(* CODESYS project 3_1_5_4.library
   Company: StroemHansen
   Title: SH_Light
   Description: Adds override function to
      FB_TwoVal_SelectOne_RTrigChange
      
      Fixes bugs in
      FB_FoldingDoorCtrl_2Pcs
      
      Replaces 3.1.5.3
   Placeholder: SH_Light
   Author: Jonas Justsen
   Version: 3.1.5.4

Project tree, tasks and I/O mapping:
  libraries: Tc2_ModbusSrv, * (Beckhoff Automation GmbH); Tc2_Standard, * (Beckhoff Automation GmbH); Tc2_System, * (Beckhoff Automation GmbH); Tc2_Utilities, * (Beckhoff Automation GmbH); Tc3_DALI, * (Beckhoff Automation GmbH)
  DUTs/
    data type E_OnMode
    data type ST_DALI_Energy
    data type ST_DALI_GrpAssignment
    data type ST_DALI_NIKOP46SetupData
    data type ST_DALI_RoomSetup
    data type ST_DALI_Sensor
    data type ST_DALI_SensorScaleMode
    data type ST_DALIButton
    data type ST_GlamoxSetup
    data type ST_GroupSort
    data type ST_LgtCmd
    data type ST_LiveData
    data type ST_LunatoneMCSetup
    data type ST_NeighborIP
    data type ST_RoomDataPLC
    data type ST_TuneData_EX
  GVLs/
    global variables DALI_Param
    global variables GVL_DALI
    global variables GVL_DALI_LatestError
  POUs/
    DALI/
      Ballast/
        function F_fDALICurve [ST]
        function F_fDALICurveRev [ST]
        function block FB_DALI_Diag [ST]: A_DALICmdAddressing, A_DALICmdAddToGroup, A_DALICmdQueryGroups, A_DALICmdQueryLampFailure, A_DALICmdQueryMissingShortAddress, A_DALICmdQueryStatus, A_ResetRoutine, A_SetAddressesToGroups, ipDALICommunication, TrySetCommunication
        function block FB_DALI_EnergyDataManagement [ST]
        function block FB_DALI_EnergyReporting [ST]: A_DALI252QueryActiveEnergy, A_DALI252QueryActiveEnergyLoadside, A_DALI252QueryActivePower, A_DALI252QueryActivePowerLoadside, A_DALI252QueryApparentEnergy, A_DALI252QueryApparentPower, A_DALI253QueryControlGearOperatingTime, A_DALI253QueryControlGearStartCounter, A_DALI253QueryLightSourceStartCounter, A_ResetRoutine, ipDALICommunication, TrySetCommunication
        function block FB_DALILgtActr_EX [ST]: A_DALICmdDirectArcPowerControl, A_DALICmdDirectArcPowerControl_Sttup, A_DALICmdDown, A_DALICmdOff, A_DALICmdQueryActualLevel, A_DALICmdQueryMaxLevel, A_DALICmdQueryMinLevel, A_DALICmdQueryPhysicalMinLevel, A_DALICmdRecallMaxLevel, A_DALICmdRecallMinLevel, A_DALICmdSetFadeRate, A_DALICmdSetFadeTime, A_DALICmdSetMaxLevel_CmdSt, A_DALICmdSetMaxLevel_Input, A_DALICmdSetMinLevel_CmdSt, A_DALICmdSetMinLevel_Input, A_DALICmdStepDown, A_DALICmdStepUp, A_DALICmdUp, A_ResetRoutine, ipDALICommunication, TrySetCommunication
        function block FB_DALILgtActr_Simple [ST]: A_DALICmdDirectArcPowerControl, A_DALICmdDirectArcPowerControl_Sttup, A_DALICmdDown, A_DALICmdOff, A_DALICmdQueryActualLevel, A_DALICmdQueryMaxLevel, A_DALICmdQueryMinLevel, A_DALICmdQueryPhysicalMinLevel, A_DALICmdRecallMaxLevel, A_DALICmdRecallMinLevel, A_DALICmdStepDown, A_DALICmdStepUp, A_DALICmdUp, A_ResetRoutine, ipDALICommunication, TrySetCommunication
        function block FB_DALILgtCfg [ST]: A_DALICmdQueryActualLevel, A_DALICmdQueryMaxLevel, A_DALICmdQueryMinLevel, A_DALICmdQueryPhysicalMinLevel, A_DALICmdSetFadeRate, A_DALICmdSetFadeTime, A_DALICmdSetMaxLevel_CmdSt, A_DALICmdSetMaxLevel_Input, A_DALICmdSetMinLevel_CmdSt, A_DALICmdSetMinLevel_Input, A_ResetRoutine, ipDALICommunication, TrySetCommunication
        function block FB_Light_Ballast [ST]: M_PrimBallast, M_SecBallast, M_SuplBallast
        function block FB_Light_SingleBallast [ST]: M_Ballast
        function block FB_MasterSelector [ST]
      Color (DT8)/
        function F_iColorMix [ST]
        function block FB_DALI_RGBWAFLight [ST]: A_DALICmdActivate_DT8, A_DALICmdTemporaryRGBDimlevel, A_DALICmdTemporaryRGBWAFControl, A_DALICmdTemporaryWAFDimlevel, A_DALIQueryColourValueAmber, A_DALIQueryColourValueBlue, A_DALIQueryColourValueFreeColor, A_DALIQueryColourValueGreen, A_DALIQueryColourValueRed, A_DALIQueryColourValueWhite, A_ResetRoutine, ipDALICommunication, TrySetCommunication
        function block FB_DALI_TcColorLight [ST]: A_DALICmdActivate_DT8, A_DALICmdSetColourTemperatureTc, A_DALIQueryColourStatus, A_DALIQueryColourTc, A_ResetRoutine, ipDALICommunication, TrySetCommunication
      DALI_Devices/
        BEG/
          function block FB_BEG_PD2N_1Pcs [ST]: A_BEG_PD2N_1
        ESYLux/
          Flat/
            function block FB_DALI_ESYLuxFlat_1Pcs [ST]: A_ESYLux_1
          function block FB_DALI_ESYLux_1Pcs [ST]: A_ESYLux_1
          function block FB_DALI_ESYLux_2Pcs [ST]: A_ESYLux_2Pcs
          function block FB_DALI_ESYLux_3Pcs [ST]: A_ESYLux_3Pcs
          function block FB_DALI_ESYLux_4Pcs [ST]: A_ESYLux_4Pcs
          function block FB_DALI_ESYLux_5Pcs [ST]: A_ESYLux_5Pcs
          function block FB_DALI_ESYLux_6Pcs [ST]: A_ESYLux_6Pcs
        Glamox/
          function block FB_DALI_GlamoxButtons [ST]: A_Sort_Event_Button1, A_Sort_Event_Button2, A_Sort_Event_Button3, A_Sort_Event_Button4, A_Sort_Event_Button5, A_Sort_Event_Button6, A_Sort_Event_Button7, A_Sort_Event_Button8
        Lunatone/
          function block FB_DALI_Lunatone_MC2_OLD [ST]: A_LunatonButton
          function block FB_DALI_Lunatone_ROT [ST]: A_LunatonRotation
          function block FB_DALI_LunatoneMC [ST]: A_Sort_Event_Button1, A_Sort_Event_Button2, A_Sort_Event_Button3, A_Sort_Event_Button4
        NIKO/
          function block FB_NIKO_P46xx_10Pcs [ST]: A_NIKO_P46xx
          function block FB_NIKO_P46xx_1Pcs [ST]: A_NIKO_P46xx_1
          function block FB_NIKO_P46xx_2Pcs [ST]: A_NIKO_P46xx
          function block FB_NIKO_P46xx_3Pcs [ST]: A_NIKO_P46xx
          function block FB_NIKO_P46xx_4Pcs [ST]: A_NIKO_P46xx
          function block FB_NIKO_P46xx_5Pcs [ST]: A_NIKO_P46xx
          function block FB_NIKO_P46xx_6Pcs [ST]: A_NIKO_P46xx
          function block FB_NIKO_P46xx_7Pcs [ST]: A_NIKO_P46xx
          function block FB_NIKO_P46xx_8Pcs [ST]: A_NIKO_P46xx
          function block FB_NIKO_P46xx_9Pcs [ST]: A_NIKO_P46xx
      FBs/
        function block FB_Short [ST]
        function block FB_ValTrig_F [ST]
      FUNs/
        function F_fScale [ST]
        function F_lrScale_EX [ST]
      Lunatone/
        function block FB_DALI_Lunatone_ROT_D2I_Mode [ST]: bEnablePosition, eEventPriorityPosition, nDeadtimerPosition, nReportTimePosition, bEnablePushButton, eEventPriorityButton, nDoubleTimerPushButton, nEventFilterPushButton, nRepeatTimerPushButton, nShortTimerPushButton, nStuckTimerPushButton, bEnableRotation, eEventPriorityRotation, nEventFilterRotation, CheckParameters, FB_init, ipDALICommunication, ParameterChanged, SetCommunication
        data type ST_ROT
      MUX/
        Timing/
          function block FB_MinOnMinOffTime [ST]
      Operators/
        function block FB_BA_Swi [ST]
        function block FB_BA_ValTrigF [ST]
        function block FB_Click [ST]
        function block FB_FileCopy [ST]
        function block FB_Ramper [ST]
      Power Control/
        function block FB_AutoTune_TcBA_EX [ST]
        function block FB_DirectLight_1Group [ST]
        function block FB_LightCtrl_1Group [ST]
        function block FB_LightCtrl_1Group_ [ST]
        function block FB_LightCtrl_1Group_OLD [ST]
        function block FB_LightCtrl_2Groups [ST]
        function block FB_LightCtrl_2Groups_Action [ST]: A_Auto, A_Manuel, A_Tuning
        function block FB_LightSwitch [ST]: A_BA_LgtSwi_ResetCommands, A_BA_LgtSwi_WaitToReset
        function block FB_SearchStartUpLevel_EX [ST]
    Folding_Doors/
      function block FB_ConnectRooms_3Pcs [ST]: A_ButtonLogic, A_OverrideLogic, A_SensorLogic
      function block FB_ConnectRooms_xPcs [ST]: A_ButtonLogic, A_OverrideLogic, A_SensorLogic
      function block FB_FoldingDoor [ST]: A_ButtonLogic, A_OverrideLogic, A_SensorLogic
      function block FB_FoldingDoorCtrl_2Pcs [ST]: A_State0, A_State1, A_State2, A_State3
    Internals/
      function block FB_FunctionType_A [ST]
    Misc/
      function F_CltsEveryBool [ST]
      function block FB_ClockPulse [ST]
      function block FB_CountOnHours [ST]
      function block FB_TwoVal_SelectOne_RTrigChange [ST]
    Modbus/
      function block FB_ReadAHPirData [ST]
    Scheduling/
      function block FB_TODScheduling [ST]
    Templates/
      function block FB_Light_Type_A [ST]: A_DaliUpdate, A_RoomFct, A_TuningProcess
      function block FB_Light_Type_B [ST]: A_DaliUpdate, A_RoomFct, A_TuningProcess
  Project Information/
    function F_GetCompany [ST]
    function F_GetTitle [ST]
    function F_GetVersion [ST]
  Version/
    global variables Global_Version
  VISUs/
*)

// DUTs/E_OnMode
TYPE E_OnMode :
(	e_ClMaxVal 				:= 0,
	e_ClMinVal 				:= 1,
	e_ClOnVal 				:= 2,
	e_ClRstVal 				:= 3
);END_TYPE

// DUTs/ST_DALI_Energy
TYPE ST_DALI_Energy :
STRUCT
	fActiveEnergy				: LREAL;
	fActiveEnergyLoadside		: LREAL;
	fActivePower				: LREAL;
	fActivePowerLoadside 		: LREAL;
	fApparentEnergy 			: LREAL;
	fApparentPower 				: LREAL;
	nControlGearOperatingTime  	: UDINT;
	nControlGearStartCounter   	: UDINT;	
	nLightSourceStartCounter   	: UDINT;
	bHasEnergyData				: BOOL;
END_STRUCT
END_TYPE

// DUTs/ST_DALI_GrpAssignment
TYPE ST_DALI_GrpAssignment :
STRUCT
	bLampPresentInNetwork: BOOL;
	bFaultOnDALIBallast : BOOL;
	bLampFailur : BOOL;
	bLampPowerOn : BOOL;
	bLimitErrVal : BOOL;
	bDimmingActive: BOOL;
	bResetState	: BOOL;
	bShortAddrMissing: BOOL;
	bPowerSupplyWasEnabled: BOOL;
	nGroups	: WORD; 	
END_STRUCT
END_TYPE

// DUTs/ST_DALI_NIKOP46SetupData
TYPE ST_DALI_NIKOP46SetupData :
STRUCT
	bInitialize						:	BOOL := TRUE;
	bQueryInputValueOccupancy			:	BOOL ;
	bQueryInputValueBrightness		:	BOOL ;
	//Parameters Motion
	bEnableInstanceOccupancy			:	BOOL := TRUE;
	eEventPriorityOccupancy			: 	E_DALIEventPriority := E_DALIEVENTPRIORITY.Middle;
	nReportTimerOccupancy				:	BYTE := 120; // Value in s, Preset manufacturer value
	nDeadtimeTimerOccupancy			:	WORD := 100; // Value in ms, Predefined Value of DALI Standard
	nHoldTimerOccupancy				:	WORD := 120; // Value in s. 
	bCancelHoldTimeOccupancy			:	BOOL := FALSE;
	nSensitivityPIRSegmentA			:	BYTE := 16#01; // Preset manufacturer value: 0 = Max, 1 = High, 2 = Low, 3 = Min, 4 = Off
	nSensitivityPIRSegmentB			:	BYTE := 16#01; // Preset manufacturer value: 0 = Max, 1 = High, 2 = Low, 3 = Min, 4 = Off
	nSensitivityPIRSegmentC			:	BYTE := 16#01; // Preset manufacturer value: 0 = Max, 1 = High, 2 = Low, 3 = Min, 4 = Off
	//Parameters Brightness
	bEnableInstanceBrightness		:	BOOL := TRUE;
	eEventPriorityBrightness		: 	E_DALIEventPriority := E_DALIEVENTPRIORITY.Middle;
	nReportTimerBrightness			:	BYTE := 120; // Value in s, Predefined Value of DALI Standard
	nDeadtimeTimerBrightness		:	WORD := 1500; // Value in ms, Predefined Value of DALI Standard
	nHysteresisBrightness			:	BYTE := 2; // Value in %
	nHysteresisMinBrightness		:	BYTE := 10; // Absolute Value, depending on the manufacturer specific resolution
	nLUXRangeBrightness				:	BYTE := 16#0; // Preset manufacturer value: 0 = Normal (0-1023 Lux, 10-bit), 1 = High (0-10360 Lux, 14-bit), 

END_STRUCT
END_TYPE

// DUTs/ST_DALI_RoomSetup
TYPE ST_DALI_RoomSetup :
STRUCT
	byShrtAdr_Prim				: BYTE:=1;	
	byGrpAdr_Prim				: BYTE :=1;	
	eMod_Prim					: E_DALIAddressType := E_DALIADDRESSTYPE.Group;

	byShrtAdr_Sec				: BYTE:=10;	
	byGrpAdr_Sec				: BYTE :=2;
	eMod_Sec					: E_DALIAddressType := E_DALIADDRESSTYPE.Group;
	
	byShrtAdr_Supl				: BYTE:=30;	
	byGrpAdr_Supl				: BYTE :=3;	
	eMod_Supl					: E_DALIAddressType := E_DALIADDRESSTYPE.Short;		

	DALI_LINE_NUM_PRIM			: BYTE := 1; //Value = 0 means the group aren't represented in the system
	DALI_LINE_NUM_SEC			: BYTE := 1; //Value = 0 means the group aren't represented in the system
	DALI_LINE_NUM_SUPL			: BYTE := 0;//Value = 0 means the group aren't represented in the system	
	
	bLocal_GlobalFadeInfo		: BOOL := TRUE;  //True = Global settings selected
	
	arrSensorScale				: ARRAY [1..12] OF ST_DALI_SensorScaleMode := [12((fMeassureMaxSensor := 1.0, fReadMaxSensor := 1.0))];
	arrSetupSensors				: ST_DALI_NIKOP46SetupData;
END_STRUCT
END_TYPE

// DUTs/ST_DALI_Sensor
TYPE ST_DALI_Sensor :
STRUCT
	fBrightness 		: REAL;
	bPrc				: BOOL;
	bQueryBrightness 	: BOOL;
	bBrightnessRead 	: BOOL;
END_STRUCT
END_TYPE

// DUTs/ST_DALI_SensorScaleMode
TYPE ST_DALI_SensorScaleMode :
STRUCT
	fMeassureMaxSensor			: REAL;
	fReadMaxSensor 				: REAL;
END_STRUCT
END_TYPE

// DUTs/ST_DALIButton
TYPE ST_DALIButton :
STRUCT
	bPressed : BOOL;
	bReleased: BOOL;
	bShortPress : BOOL;
	bDoublePress : BOOL;
	bLongPressStart : BOOL;
	bLongPressRepeat : BOOL;
	bLongPressStop : BOOL;
	bButtonFree : BOOL;
END_STRUCT
END_TYPE

// DUTs/ST_GlamoxSetup
TYPE ST_GlamoxSetup :
STRUCT
	arrEnablePushButton : ARRAY [1..8] OF BOOL;
	arrEventPriorityPushButton: ARRAY [1..8] OF E_DALIEventPriority := [8(E_DALIEVENTPRIORITY.MiddleLow)];
	nDoubleTimerPushButton: UINT := 250; 	// Time in MS
	nEventFilterPushButton: ARRAY [1..8] OF BYTE := [8(2#10000111)];	  
												// BIT 0 - Button Released, The push button was released.
												// Bit 1 - Button Pressed, The push button was pressed.
												// Bit 2 - Short Press, The push button was pressed and quickly released again without being pressed again (short button press).
												// Bit 3 - Double Press, The push button was pressed, released and quickly pressed again (double button press).
												// Bit 4 - Long Press Start, The push button was pressed without being released in between times (long button press).
												// Bit 5 - Long Press Repeat, If the push button was pressed for a long period (Long Press Start) without being released in between times, this event is sent at regular intervals.
												// Bit 6 - Long Press Stop, This event is sent if the push button is released after a long button press.
												// Bit 7 - Button Free / Button Stuck, If the push button is pressed for a very long time, it is assumed that it has stuck and the Button Stuck event is sent. Button Free is sent when the push button is detected as not pressed again.
	nRepeatTimerPushButton: UINT := 160; 	// Interval (100…2000 ms) of repetitive events in the case of a long button press.
	nShortTimerPushButton: UINT := 500;		// Time (tShortMin...5100 ms) to distinguish between a long and a short button press. tShortMin is a manufacturer-specific value.
	nStuckTimerPushButton: BYTE := 20; 		// Time (5…255 s) after whose expiry the push button no longer represents a long button press. The push button is stuck.

END_STRUCT
END_TYPE

// DUTs/ST_GroupSort
TYPE ST_GroupSort :
STRUCT
	arrAddrInGroups			: ARRAY[0..63, 0..15] OF BOOL;
	arrAddressesInEachGroup : ARRAY[0..15, 0..63] OF BYTE;
END_STRUCT
END_TYPE

// DUTs/ST_LgtCmd
TYPE ST_LgtCmd :
STRUCT
	bOff				: BOOL;	
	bClMinCtrlVal		: BOOL;
	bClMaxCtrlVal		: BOOL;
	bClOnVal			: BOOL;
	lrOnVal				: REAL;
	bClRstVal			: BOOL;
	bSetCtrlValDct		: BOOL;
	fSetCtrlValDct		: REAL;
	bChgMinCtrlVal		: BOOL;
    fChgMinCtrlVal		: REAL;
    bChgMaxCtrlVal		: BOOL;
    fChgMaxCtrlVal		: REAL;
    bDimUp				: BOOL;
    bDimDwn				: BOOL;
    bStpUp				: BOOL;
    bStpDwn				: BOOL;
END_STRUCT
END_TYPE

// DUTs/ST_LiveData
TYPE ST_LiveData :
STRUCT
// Light live data
	bLightON_Zone_1 		: BOOL;
	bLightOFF_Zone_1 		: BOOL;
	bLightAuto_Zone_1 		: BOOL;
	bLightManuel_Zone_1 	: BOOL;
	bLightON_Zone_2 		: BOOL;
	bLightOFF_Zone_2 		: BOOL;
	bLightAuto_Zone_2 		: BOOL;
	bLightManuel_Zone_2 	: BOOL;	
	
// Live data PIR sensor
	stPir					: ST_DALI_Sensor;
	bRoomOccupied			: BOOL;
	
//Alarm data
	bAlarmEnabled 			: BOOL;
END_STRUCT
END_TYPE

// DUTs/ST_LunatoneMCSetup
TYPE ST_LunatoneMCSetup :
STRUCT
	arrEnablePushButton : ARRAY [1..4] OF BOOL;
	arrEventPriorityPushButton: ARRAY [1..4] OF E_DALIEventPriority := [4(E_DALIEVENTPRIORITY.MiddleLow)];
	nDoubleTimerPushButton: UINT := 250; 	// Time in MS
	nEventFilterPushButton: ARRAY [1..4] OF BYTE := [4(2#10000111)];	  
												// BIT 0 - Button Released, The push button was released.
												// Bit 1 - Button Pressed, The push button was pressed.
												// Bit 2 - Short Press, The push button was pressed and quickly released again without being pressed again (short button press).
												// Bit 3 - Double Press, The push button was pressed, released and quickly pressed again (double button press).
												// Bit 4 - Long Press Start, The push button was pressed without being released in between times (long button press).
												// Bit 5 - Long Press Repeat, If the push button was pressed for a long period (Long Press Start) without being released in between times, this event is sent at regular intervals.
												// Bit 6 - Long Press Stop, This event is sent if the push button is released after a long button press.
												// Bit 7 - Button Free / Button Stuck, If the push button is pressed for a very long time, it is assumed that it has stuck and the Button Stuck event is sent. Button Free is sent when the push button is detected as not pressed again.
	nRepeatTimerPushButton: UINT := 160; 	// Interval (100…2000 ms) of repetitive events in the case of a long button press.
	nShortTimerPushButton: UINT := 500;		// Time (tShortMin...5100 ms) to distinguish between a long and a short button press. tShortMin is a manufacturer-specific value.
	nStuckTimerPushButton: BYTE := 20; 		// Time (5…255 s) after whose expiry the push button no longer represents a long button press. The push button is stuck.

END_STRUCT
END_TYPE

// DUTs/ST_NeighborIP
TYPE ST_NeighborIP :
STRUCT
	sPLCName	: STRING(5);
	sIP				: STRING(15);
	IsNeighbor	: BOOL := FALSE;
END_STRUCT
END_TYPE

// DUTs/ST_RoomDataPLC
TYPE ST_RoomDataPLC :
STRUCT
	bPirActive			:	BOOL;
	uiPirOffDelayTime	:	UINT;
	uiActLuxLevel		:	UINT;
	uiSpLuxLevel		:	UINT;
	uiActLightLevelPct	:	UINT;
	uiBallastOnHours	:	UINT;
	
	uiPirDimDelayTime	:	UINT;
	uiSpDimLuxLevel		:	UINT;
END_STRUCT
END_TYPE

// DUTs/ST_TuneData_EX
TYPE ST_TuneData_EX :
STRUCT
	arrLuxLevels : ARRAY [0..20] OF REAL;
	bTunnigDone : BOOL;
END_STRUCT
END_TYPE

// POUs/DALI/Lunatone/ST_ROT
TYPE ST_ROT :
STRUCT
	nPos 		: BYTE;

	bCW 		: BOOL;
	bCCW 		: BOOL;
	bStopped 	: BOOL;
	
	bPressed 	: BOOL;
	bReleased 	: BOOL;
END_STRUCT
END_TYPE

// GVLs/DALI_Param
VAR_GLOBAL CONSTANT
	tOutTuneDelay						: TIME := T#15S;
	eGlobalFadeTime					: E_DALIFadeTime:= E_DALIFadeTime.T02000ms;
	MAX_DALIV2_LINES			: BYTE := 6;
	nPlcTaskCycleTimeInMS		: UDINT:= 40;
	nDimCmdCycleTimeFactor	: UDINT:= 2;
	byMaxNumOfFoldingDoors	: BYTE := 2;
END_VAR

// GVLs/GVL_DALI
VAR_GLOBAL

	arrbBlockDTR 			: ARRAY[1..DALI_Param.MAX_DALIV2_LINES] OF BOOL;
	g_arrDiagnosisRunOnce	: ARRAY [1..DALI_Param.MAX_DALIV2_LINES] OF BOOL;
	g_arrGrpAssignment		: ARRAY[1..DALI_Param.MAX_DALIV2_LINES, 0..63] OF ST_DALI_GrpAssignment;
	g_arrAddrInGroups		: ARRAY[1..DALI_Param.MAX_DALIV2_LINES] OF ST_GroupSort;
	{attribute 'OPC.UA.DA' := '1'}
	{attribute 'OPC.UA.DA.Access' := '1'}
	{attribute 'OPC.UA.DA.StructuredType' := '1'}
	g_arrEnergyData			: ARRAY[1..DALI_Param.MAX_DALIV2_LINES, 0..63] OF ST_DALI_Energy ;
END_VAR

// GVLs/GVL_DALI_LatestError
{attribute 'qualified_only'}
VAR_GLOBAL
	arrLineShrtAddr		: ARRAY[1..DALI_Param.MAX_DALIV2_LINES] OF BYTE := [DALI_Param.MAX_DALIV2_LINES(255)];
END_VAR

// Version/Global_Version
{attribute 'TcGenerated'}
{attribute 'no-analysis'}
{attribute 'linkalways'}
// This function has been automatically generated from the project information.
VAR_GLOBAL CONSTANT
	{attribute 'const_non_replaced'}
	stLibVersion_SH_Light : ST_LibVersion := (iMajor := 3, iMinor := 1, iBuild := 5, iRevision := 4, nFlags := 0, sVersion := '3.1.5.4');
END_VAR

// POUs/DALI/Ballast/F_fDALICurve
FUNCTION F_fDALICurve : REAL
VAR_INPUT
	fPctSatsIn: REAL;
END_VAR
VAR
	fLOGSats: REAL;
	fLOG10: REAL;
	fConstantValue: REAL := 84.3333333333333;
END_VAR


IF fPctSatsIn<=0 THEN
	F_fDALICurve:= 0;
ELSE
	fLOGSats:= LOG(fPctSatsIn);
	fLOG10:=LREAL_TO_REAL(LOG(10));

	F_fDALICurve:= (((fLOGSats/fLOG10)+1) * fConstantValue)+1;

	IF fPctSatsIn>=100 THEN
		F_fDALICurve:= 254;
	END_IF
END_IF

END_FUNCTION

// POUs/DALI/Ballast/F_fDALICurveRev
FUNCTION F_fDALICurveRev : REAL
VAR_INPUT
	fDALIValue: REAL;
END_VAR
VAR
	fConstantValue: REAL := 84.3333333333333;
END_VAR


IF fDALIValue<=0 THEN
	F_fDALICurveRev:= 0;
ELSE
	F_fDALICurveRev:=LREAL_TO_REAL((EXPT(10, (fDALIValue/fConstantValue)-(1/fConstantValue)-1)));

	IF fDALIValue>=254 THEN
		F_fDALICurveRev:= 100;
	END_IF
END_IF

END_FUNCTION

// POUs/DALI/Ballast/FB_DALI_Diag
FUNCTION_BLOCK FB_DALI_Diag
VAR_INPUT	
	bReInit: BOOL;
	bErrorFromSystem 				: BOOL;
	DALI_LINE_NUM					: BYTE := 1;
END_VAR
VAR_OUTPUT
	bMissingShortAddress: BOOL;
	bOneDaliBallastMissing: BOOL;
	bSeveralMissingShortAddress: BOOL;
	bInitialized	: BOOL;
	bBusy: BOOL;
	nErrorId: UDINT;
	bErr: BOOL;
END_VAR
VAR
	ipCommunication					: I_DALICommunication;
	ipCommunicationPreset			: I_DALICommunication;
	fbDALI102QueryStatus			: FB_DALI102QueryStatus(0);
	fbDALI102QueryGroups			: FB_DALI102QueryGroups(0);
	fbDALI102QueryLampFailure		: FB_DALI102QueryLampFailure(0);
	fbDALI102Addressing				: FB_DALI102Addressing(0);
	fbDALI102AddToGroup				: FB_DALI102AddToGroup(0);
	fbDALI102QueryMissingShortAddress	: FB_DALI102QueryMissingShortAddress(0);
	

	nAddress						: BYTE;
	eAddrType						: E_DALIAddressType := E_DALIADDRESSTYPE.Short;
	eCmdPrio						: E_DALICommandPriority := E_DALICommandPriority.Low;
	nStepStatus						: INT;

	fbDelayBeforeNextTest			: TON;
	fbDelayCheckLine				: TON;
	nStepBeforeErr					: INT;
	nDaliBalastStatus				: BYTE;
	nIdxAdr							: BYTE;
	nIdxGrp							: BYTE;
	arrIDXCount						: ARRAY[0..15] OF BYTE;

	arrGroupAssignment: ARRAY[0..63] OF WORD;
	bActionBusy: BOOL;

	nGroup: BYTE;
	nAddrMissing: BYTE;

	nSearchIdx: INT;
	arrDALIBallastInNetwork: ARRAY[0..63] OF byte;
	nBallastIndex: INT;
	nGroupsTheBallastAssign: ARRAY[0..15] OF BOOL;
	iGrpSearch: byte;
	fbReinit_RTrig: R_Trig;
END_VAR

{region "initialize the outputs"}
IF (NOT bInitialized) THEN
	THIS^.TrySetCommunication();		 
	bBusy := TRUE;
	nErrorId := 0;
	bErr := FALSE;
	bInitialized := TRUE;
END_IF
	 
//Reinit system
fbReinit_RTrig(CLK:=bReInit);	

IF fbReinit_RTrig.Q THEN
	bInitialized := FALSE;
END_IF 
{endregion}


{region "check parameters"}
IF (ipCommunication = 0) THEN
	bErr := TRUE;
	nErrorId := TC_EVENTS.TcDALIEventClass.TheInterfaceToTheCommunicationBufferIsNotInitialized.nEventId;
	nStepStatus := 0;
END_IF
IF ((eAddrType <> E_DALIAddressType.Short) AND (eAddrType <> E_DALIAddressType.Group) AND (eAddrType <> E_DALIAddressType.Broadcast) AND (eAddrType <> E_DALIAddressType.BroadcastUnaddr)) THEN
	bErr := TRUE;
	nErrorId := TC_EVENTS.TcDALIEventClass.ParameterAddressTypeLiesOutsideOfTheValidRange.nEventId;
	nStepStatus := 0;
END_IF
IF ((eAddrType = E_DALIAddressType.Short) AND (nAddress > 63)) THEN
	bErr := TRUE;
	nErrorId := TC_EVENTS.TcDALIEventClass.ParameterAddressIsAShortAddressAndLiesOutsideOfTheValidRange.nEventId;
	nStepStatus := 0;
END_IF

IF ( nAddress> 63) THEN
	bErr := TRUE;
	nErrorId := 16#8000; // custom error code: Parameter byShrtAdr lies outside of the valid range
	nStepStatus := 0;
END_IF
{endregion}

CASE nStepStatus OF

0: //Init state		

	IF NOT g_arrDiagnosisRunOnce[DALI_LINE_NUM] THEN
		nStepStatus:= 1000;
		A_ResetRoutine();
		bBusy := TRUE;	 
	ELSE
		fbDelayCheckLine(IN:= TRUE, PT:=T#1H);
		IF fbDelayCheckLine.Q  AND NOT bOneDaliBallastMissing THEN
			A_ResetRoutine();
			nStepStatus:= 100;
			fbDelayCheckLine(IN:= FALSE);
			bBusy := TRUE;
			bOneDaliBallastMissing := FALSE;	 
		ELSIF fbDelayCheckLine.Q  AND bOneDaliBallastMissing THEN
			A_ResetRoutine();
			nStepStatus:= 300;
			fbDelayCheckLine(IN:= FALSE);
			bBusy := TRUE;	 
		ELSIF bErrorFromSystem THEN
			A_ResetRoutine();
			nStepStatus:= 200;
			fbDelayCheckLine(IN:= FALSE);
			bBusy := TRUE;	 	 
		END_IF
	END_IF

// CYCLICK CHECKS FOR DALI LAMPFALIURE
100:	//Check if somthing wrong in DALI line

	A_DALICmdQueryLampFailure();
	IF NOT bActionBusy	THEN
		IF bErr	THEN
			nStepStatus:= 0;
			bBusy := FALSE;		 
		ELSE
			nStepStatus:= 101;
		END_IF
	 END_IF
		  
101:	
	 
	IF NOT bActionBusy	THEN
		IF bErr	THEN
			nStepStatus:= 0;
		ELSE
			IF fbDALI102QueryLampFailure.bLampFailure THEN
				nBallastIndex := 0;
				nStepStatus:= 200;
				bBusy := FALSE;		 
			ELSE
				nStepStatus:= 0;
				bBusy := FALSE;
			END_IF	 
			
		END_IF
	END_IF


200: //Finding the lamp with error
 	//Start init routinge for checking the DALI bus for ballast and group assignment
		nStepStatus:= 201;
		A_ResetRoutine();	 
		bActionBusy:= FALSE;
		nBallastIndex := 0;	 
		nAddress := arrDALIBallastInNetwork[nBallastIndex];			//Starting the serach from first addr in lamp array -->

201:	//Start query which ballast are present on the bus
	
	IF nAddress <> 99 THEN	 
		A_DALICmdQueryStatus();
		IF NOT bActionBusy THEN
			IF bErr	THEN
				nStepBeforeErr:= nStepStatus;
				A_ResetRoutine();	 
				nStepStatus:= 300 ;	//Lamp found, please see when new ballast are attached
				nAddrMissing := arrDALIBallastInNetwork[nBallastIndex];	 
				bOneDaliBallastMissing := TRUE;	 
			ELSE
				nStepStatus:= 210; 	//This lamp are still OK, please check the next ballast in network
			END_IF
		END_IF
	ELSE
		 nStepStatus:= 210; 	//This lamp are still OK, please check the next ballast in network
	END_IF		  
 
210: //Add one to DALI addreees for checking
	
	IF nBallastIndex < 63 THEN
		bErr := FALSE;
		nBallastIndex := nBallastIndex + 1;
		nAddress := arrDALIBallastInNetwork[nBallastIndex];			//Select next address from list
		IF nAddress > 63 THEN
			nAddress := 63;	 
			nStepStatus:= 211 ;		 
		ELSE
			nStepStatus := 201;
		END_IF		  
	ELSE
		IF bErrorFromSystem	THEN
				 
			nStepStatus:= 300;
		ELSE
			nBallastIndex := 0;
			nStepStatus:= 0 ;
			bBusy := FALSE ; 
		END_IF		 
	END_IF	

211:
	 nStepStatus:= 210 ;	
		  
300:	//Start to check if new Unaddressed ballast are present
	A_DALICmdQueryMissingShortAddress();
	IF NOT bActionBusy THEN
		IF bErr	THEN
			nStepBeforeErr:= nStepStatus;
			nStepStatus:= 301 ;	//Lamp found, please see when new ballast are attached
		ELSE
			IF bMissingShortAddress THEN	 
				nStepStatus:= 400; 	//This lamp are still OK, please check the next ballast in network
				A_ResetRoutine();
			ELSIF bSeveralMissingShortAddress THEN
				nStepStatus := 0;
			ELSIF NOT bMissingShortAddress AND NOT bSeveralMissingShortAddress THEN
				nStepStatus := 1000;	 
			END_IF			 
		END_IF
		
	END_IF

301:	//Wait before test again  
	fbDelayBeforeNextTest(IN:=TRUE , PT:= T#1M , Q=> , ET=> );
	IF fbDelayBeforeNextTest.Q THEN
		A_ResetRoutine();
		fbDelayBeforeNextTest(IN:=FALSE);	 
		nStepStatus:= 300;
	END_IF


400: //Set DALI Address to ballast without addresse

	A_DALICmdAddressing();
	IF NOT bActionBusy THEN
		IF bErr	THEN
			nStepBeforeErr:= nStepStatus;
			nStepStatus:= 0 ;
			bOneDaliBallastMissing := TRUE;	 
		ELSE
			nStepStatus:= 401; 	//This lamp are still OK, please check the next ballast in network
 			nGroupsTheBallastAssign[0]:=GVL_DALI.g_arrGrpAssignment[DALI_LINE_NUM, nAddrMissing].nGroups.0;
			nGroupsTheBallastAssign[1]:=GVL_DALI.g_arrGrpAssignment[DALI_LINE_NUM, nAddrMissing].nGroups.1;
			nGroupsTheBallastAssign[2]:=GVL_DALI.g_arrGrpAssignment[DALI_LINE_NUM, nAddrMissing].nGroups.2;
			nGroupsTheBallastAssign[3]:=GVL_DALI.g_arrGrpAssignment[DALI_LINE_NUM, nAddrMissing].nGroups.3;
			nGroupsTheBallastAssign[4]:=GVL_DALI.g_arrGrpAssignment[DALI_LINE_NUM, nAddrMissing].nGroups.4;
			nGroupsTheBallastAssign[5]:=GVL_DALI.g_arrGrpAssignment[DALI_LINE_NUM, nAddrMissing].nGroups.5;
			nGroupsTheBallastAssign[6]:=GVL_DALI.g_arrGrpAssignment[DALI_LINE_NUM, nAddrMissing].nGroups.6;
			nGroupsTheBallastAssign[7]:=GVL_DALI.g_arrGrpAssignment[DALI_LINE_NUM, nAddrMissing].nGroups.7;
			nGroupsTheBallastAssign[8]:=GVL_DALI.g_arrGrpAssignment[DALI_LINE_NUM, nAddrMissing].nGroups.8;
			nGroupsTheBallastAssign[9]:=GVL_DALI.g_arrGrpAssignment[DALI_LINE_NUM, nAddrMissing].nGroups.9;
			nGroupsTheBallastAssign[10]:=GVL_DALI.g_arrGrpAssignment[DALI_LINE_NUM, nAddrMissing].nGroups.10;
			nGroupsTheBallastAssign[11]:=GVL_DALI.g_arrGrpAssignment[DALI_LINE_NUM, nAddrMissing].nGroups.11;
			nGroupsTheBallastAssign[12]:=GVL_DALI.g_arrGrpAssignment[DALI_LINE_NUM, nAddrMissing].nGroups.12;
			nGroupsTheBallastAssign[13]:=GVL_DALI.g_arrGrpAssignment[DALI_LINE_NUM, nAddrMissing].nGroups.13;
			nGroupsTheBallastAssign[14]:=GVL_DALI.g_arrGrpAssignment[DALI_LINE_NUM, nAddrMissing].nGroups.14;
			nGroupsTheBallastAssign[15]:=GVL_DALI.g_arrGrpAssignment[DALI_LINE_NUM, nAddrMissing].nGroups.15;
			iGrpSearch := 0;	 
		END_IF
		
	END_IF

401: //Check for writing group assignemnt to the ballast
	
	IF 	nGroupsTheBallastAssign[iGrpSearch] THEN
		nGroup := iGrpSearch;
		A_ResetRoutine();
		nStepStatus := 410 ;	 
	ELSE		 
	 	nStepStatus := 402;
	END_IF
		 
402:	
	IF iGrpSearch<15 THEN
 		iGrpSearch := iGrpSearch + 1 ;
		nStepStatus := 401 ;
	ELSE
		nStepStatus := 0 ;
	END_IF

410:
	A_DALICmdAddToGroup();
	IF NOT bActionBusy THEN
		IF bErr	THEN
			nStepBeforeErr:= nStepStatus;
			nStepStatus:= 0 ;	//Lamp found, please see when new ballast are attached
		ELSE
				IF iGrpSearch<15 THEN
 					iGrpSearch := iGrpSearch + 1 ;
					nStepStatus := 401 ;
				ELSE
					nStepStatus := 300 ;	//Chekck again that All are fine for now
					A_ResetRoutine();
					iGrpSearch := 0;	 
				END_IF
		END_IF
	END_IF
	 
(* - - - - - - - - - - - - - - - - - - - - - - - - *)
(*Init Device-Routine*)

1000: //Start init routinge for checking the DALI bus for ballast and group assignment
		nStepStatus:= 1001;
		A_ResetRoutine();	 
		bActionBusy:= FALSE;
		bErr := FALSE;	 
		MEMSET(ADR(arrDALIBallastInNetwork), 99, SIZEOF(arrDALIBallastInNetwork));
		nAddress := 0;			//Starting the serach from address 0 -->
		GVL_DALI.g_arrGrpAssignment[DALI_LINE_NUM, nAddress].bLampPresentInNetwork:= FALSE;
1001:	//Start query which ballast are present on the bus
	
	A_DALICmdQueryStatus();
	IF NOT bActionBusy THEN
		IF bErr	THEN
			nStepBeforeErr:= nStepStatus;
			GVL_DALI.g_arrGrpAssignment[DALI_LINE_NUM, nAddress].bLampPresentInNetwork:= FALSE;	 
			nStepStatus:= 1004 ;	//Automatically jump to see if more addresses need to be tested
		ELSE
			GVL_DALI.g_arrGrpAssignment[DALI_LINE_NUM, nAddress].bLampPresentInNetwork:= TRUE;
			nStepStatus:= 1002;
		END_IF
		
	END_IF

1002: 
	
	GVL_DALI.g_arrGrpAssignment[DALI_LINE_NUM, nAddress].bFaultOnDALIBallast:= nDaliBalastStatus.0;
	GVL_DALI.g_arrGrpAssignment[DALI_LINE_NUM, nAddress].bLampFailur := nDaliBalastStatus.1;
	GVL_DALI.g_arrGrpAssignment[DALI_LINE_NUM, nAddress].bLampPowerOn:= nDaliBalastStatus.2;
	GVL_DALI.g_arrGrpAssignment[DALI_LINE_NUM, nAddress].bLimitErrVal := nDaliBalastStatus.3;
	GVL_DALI.g_arrGrpAssignment[DALI_LINE_NUM, nAddress].bDimmingActive:= nDaliBalastStatus.4;
	GVL_DALI.g_arrGrpAssignment[DALI_LINE_NUM, nAddress].bResetState:= nDaliBalastStatus.5;
	GVL_DALI.g_arrGrpAssignment[DALI_LINE_NUM, nAddress].bShortAddrMissing:= nDaliBalastStatus.6;
	GVL_DALI.g_arrGrpAssignment[DALI_LINE_NUM, nAddress].bPowerSupplyWasEnabled:= nDaliBalastStatus.7;
	
	nStepStatus:= 1003;

1003: //Test which group each ballast are placed
	A_DALICmdQueryGroups();
	IF NOT bActionBusy	THEN
		IF bErr	THEN
			nStepStatus:= 1004;
		ELSE
			nStepStatus:= 1004; //TODO
		END_IF
	END_IF

1004: //Add one to DALI addreees for checking
	
	IF nAddress < 63 THEN
		bErr := FALSE;
		nAddress := nAddress + 1;
		nDaliBalastStatus := 255;	 
		nStepStatus:= 1001 ;	
		GVL_DALI.g_arrGrpAssignment[DALI_LINE_NUM, nAddress].bLampPresentInNetwork:= FALSE;
	ELSE
		A_ResetRoutine();	 
	 	nAddress := 0;
		A_SetAddressesToGroups();	 
		g_arrDiagnosisRunOnce[DALI_LINE_NUM]:= TRUE;	 
		nStepStatus:= 1005 ;
		bBusy := FALSE ;
	END_IF


1005: //Ending find the number of normal ballast in network and prepare for further test later

	FOR nSearchIdx := 0 TO 63 BY 1 DO
		IF GVL_DALI.g_arrGrpAssignment[DALI_LINE_NUM, nSearchIdx].bLampPresentInNetwork	THEN
			arrDALIBallastInNetwork[nBallastIndex]:= INT_TO_BYTE(nSearchIdx);
			nBallastIndex := nBallastIndex + 1;	
		END_IF 
	END_FOR
	nBallastIndex := 0;	 
	nStepStatus:= 0 ;
	
ELSE
	nStepStatus:=0;
END_CASE

ACTION A_DALICmdAddressing:


	bActionBusy	:= TRUE;

	fbDALI102Addressing(
		bError=> , 
		ipResultMessage=> , 
		bStart:= TRUE, 
		nStartWithShortAddress:= nAddrMissing, 
		nOptions:= Tc3_DALI.GVL.cOpticalFeedback, 
		bBusy=> , 
		nAddressedDevices=> );
	
	
	IF (NOT fbDALI102Addressing.bBusy) THEN
		IF fbDALI102Addressing.bError THEN
			bErr := TRUE;
			nErrorId := fbDALI102Addressing.ipResultMessage.nEventId;
		END_IF
		bActionBusy		:= FALSE;
		fbDALI102Addressing(bStart:= FALSE);
	END_IF
END_ACTION

ACTION A_DALICmdAddToGroup:


	bActionBusy	:= TRUE;

	fbDALI102AddToGroup(
		bError=> , 
		ipResultMessage=> , 
		bStart:= TRUE, 
		nAddress:= nAddress, 
		eAddressType:= E_DALIAddressType.Short, 
		eCommandPriority:= E_DALICommandPriority.Middle , 
		bBusy=> , 
		nGroup:= nGroup);
	
	IF (NOT fbDALI102AddToGroup.bBusy) THEN
		IF fbDALI102AddToGroup.bError THEN
			bErr := TRUE;
			nErrorId := fbDALI102AddToGroup.ipResultMessage.nEventId;
		END_IF
		bActionBusy		:= FALSE;
		fbDALI102AddToGroup(bStart:= FALSE);
	END_IF
END_ACTION

ACTION A_DALICmdQueryGroups:

	bActionBusy	:= TRUE;

	
	fbDALI102QueryGroups(bStart:= TRUE, 
		nAddress:= nAddress, 
		eAddressType:= eAddrType, 
		eCommandPriority:= eCmdPrio,
		nGroups=> GVL_DALI.g_arrGrpAssignment[DALI_LINE_NUM, nAddress].nGroups);


	IF NOT fbDALI102QueryGroups.bBusy	THEN
		IF	fbDALI102QueryGroups.bError	THEN
			bErr     	:= TRUE;
			nErrorId := fbDALI102QueryGroups.ipResultMessage.nEventId;
		END_IF
		bActionBusy		:= FALSE;
		fbDALI102QueryGroups(bStart:= FALSE );
	END_IF
END_ACTION

ACTION A_DALICmdQueryLampFailure:

	bActionBusy	:= TRUE;

	
	fbDALI102QueryLampFailure(
		bStart:= TRUE , 
		eAddressType:= E_DALIAddressType.Broadcast, 
		eCommandPriority:=eCmdPrio , 
		bBusy=> , 
		bLampFailure=>);



	IF NOT fbDALI102QueryLampFailure.bBusy	THEN
		IF	fbDALI102QueryLampFailure.bError	THEN
			bErr     	:= TRUE;
			nErrorId := fbDALI102QueryLampFailure.ipResultMessage.nEventId;
		END_IF
		bActionBusy		:= FALSE;
		fbDALI102QueryLampFailure(bStart:= FALSE );
	END_IF
END_ACTION

ACTION A_DALICmdQueryMissingShortAddress:

	bActionBusy	:= TRUE;

	
	fbDALI102QueryMissingShortAddress(
		bStart:= TRUE , 
		eAddressType:= E_DALIAddressType.Broadcast, 
		eCommandPriority:=eCmdPrio , 
		bBusy=> , 
		bMissingShortAddress=>bMissingShortAddress);



	IF NOT fbDALI102QueryMissingShortAddress.bBusy	THEN
		IF	fbDALI102QueryMissingShortAddress.bError	THEN
			bErr     	:= TRUE;
			nErrorId := fbDALI102QueryMissingShortAddress.ipResultMessage.nEventId;
		END_IF
		IF fbDALI102QueryMissingShortAddress.ipResultMessage.nEventId = 27 THEN
			bSeveralMissingShortAddress:= TRUE;
		ELSE
			bSeveralMissingShortAddress:= FALSE;
		END_IF

		bActionBusy		:= FALSE;
		fbDALI102QueryMissingShortAddress(bStart:= FALSE );
	END_IF
END_ACTION

ACTION A_DALICmdQueryStatus:

	bActionBusy	:= TRUE;

	
	fbDALI102QueryStatus(
		bError=> , 
		ipResultMessage=> , 
		bStart:= TRUE, 
		nAddress:= nAddress, 
		eAddressType:= eAddrType, 
		eCommandPriority:= eCmdPrio, 
		bBusy=> , 
		nStatus=>nDaliBalastStatus );


	IF NOT fbDALI102QueryStatus.bBusy	THEN
		IF	fbDALI102QueryStatus.bError	THEN
			bErr     	:= TRUE;
			nErrorId := fbDALI102QueryStatus.ipResultMessage.nEventId;
		END_IF
		bActionBusy		:= FALSE;
		fbDALI102QueryStatus(bStart:= FALSE );
	END_IF
END_ACTION

ACTION A_ResetRoutine:
	bErr     	:= FALSE;
	nErrorId 	:= 0;

	fbDALI102QueryStatus(bStart:= FALSE );
	fbDALI102QueryGroups(bStart:= FALSE );
	fbDALI102QueryLampFailure(bStart:= FALSE );
	fbDALI102Addressing(bStart:= FALSE );
	fbDALI102AddToGroup(bStart:= FALSE );
	fbDALI102QueryMissingShortAddress(bStart:= FALSE );
END_ACTION

ACTION A_SetAddressesToGroups:

//Reset the sorting table before fill with new data
MEMSET(ADR(GVL_DALI.g_arrAddrInGroups[DALI_LINE_NUM]), 255, SIZEOF(GVL_DALI.g_arrAddrInGroups[DALI_LINE_NUM]));
MEMSET(ADR(arrIDXCount),0, SIZEOF(arrIDXCount));

//Start sorting out Bit algoritme for Group assign pr. ballast.
FOR nIdxAdr := 0 TO 63 DO
	arrGroupAssignment[nIdxAdr]:=GVL_DALI.g_arrGrpAssignment[DALI_LINE_NUM, nIdxAdr].nGroups;
	
	GVL_DALI.g_arrAddrInGroups[DALI_LINE_NUM].arrAddrInGroups[nIdxAdr, 0] := GVL_DALI.g_arrGrpAssignment[DALI_LINE_NUM, nIdxAdr].nGroups.0;
	GVL_DALI.g_arrAddrInGroups[DALI_LINE_NUM].arrAddrInGroups[nIdxAdr, 1] := GVL_DALI.g_arrGrpAssignment[DALI_LINE_NUM, nIdxAdr].nGroups.1;
	GVL_DALI.g_arrAddrInGroups[DALI_LINE_NUM].arrAddrInGroups[nIdxAdr, 2] := GVL_DALI.g_arrGrpAssignment[DALI_LINE_NUM, nIdxAdr].nGroups.2;
	GVL_DALI.g_arrAddrInGroups[DALI_LINE_NUM].arrAddrInGroups[nIdxAdr, 3] := GVL_DALI.g_arrGrpAssignment[DALI_LINE_NUM, nIdxAdr].nGroups.3;
	GVL_DALI.g_arrAddrInGroups[DALI_LINE_NUM].arrAddrInGroups[nIdxAdr, 4] := GVL_DALI.g_arrGrpAssignment[DALI_LINE_NUM, nIdxAdr].nGroups.4;
	GVL_DALI.g_arrAddrInGroups[DALI_LINE_NUM].arrAddrInGroups[nIdxAdr, 5] := GVL_DALI.g_arrGrpAssignment[DALI_LINE_NUM, nIdxAdr].nGroups.5;
	GVL_DALI.g_arrAddrInGroups[DALI_LINE_NUM].arrAddrInGroups[nIdxAdr, 6] := GVL_DALI.g_arrGrpAssignment[DALI_LINE_NUM, nIdxAdr].nGroups.6;
	GVL_DALI.g_arrAddrInGroups[DALI_LINE_NUM].arrAddrInGroups[nIdxAdr, 7] := GVL_DALI.g_arrGrpAssignment[DALI_LINE_NUM, nIdxAdr].nGroups.7;
	GVL_DALI.g_arrAddrInGroups[DALI_LINE_NUM].arrAddrInGroups[nIdxAdr, 8] := GVL_DALI.g_arrGrpAssignment[DALI_LINE_NUM, nIdxAdr].nGroups.8;
	GVL_DALI.g_arrAddrInGroups[DALI_LINE_NUM].arrAddrInGroups[nIdxAdr, 9] := GVL_DALI.g_arrGrpAssignment[DALI_LINE_NUM, nIdxAdr].nGroups.9;
	GVL_DALI.g_arrAddrInGroups[DALI_LINE_NUM].arrAddrInGroups[nIdxAdr, 10] := GVL_DALI.g_arrGrpAssignment[DALI_LINE_NUM, nIdxAdr].nGroups.10;
	GVL_DALI.g_arrAddrInGroups[DALI_LINE_NUM].arrAddrInGroups[nIdxAdr, 11] := GVL_DALI.g_arrGrpAssignment[DALI_LINE_NUM, nIdxAdr].nGroups.11;
	GVL_DALI.g_arrAddrInGroups[DALI_LINE_NUM].arrAddrInGroups[nIdxAdr, 12] := GVL_DALI.g_arrGrpAssignment[DALI_LINE_NUM, nIdxAdr].nGroups.12;
	GVL_DALI.g_arrAddrInGroups[DALI_LINE_NUM].arrAddrInGroups[nIdxAdr, 13] := GVL_DALI.g_arrGrpAssignment[DALI_LINE_NUM, nIdxAdr].nGroups.13;
	GVL_DALI.g_arrAddrInGroups[DALI_LINE_NUM].arrAddrInGroups[nIdxAdr, 14] := GVL_DALI.g_arrGrpAssignment[DALI_LINE_NUM, nIdxAdr].nGroups.14;
	GVL_DALI.g_arrAddrInGroups[DALI_LINE_NUM].arrAddrInGroups[nIdxAdr, 15] := GVL_DALI.g_arrGrpAssignment[DALI_LINE_NUM, nIdxAdr].nGroups.15;
END_FOR

FOR nIdxGrp:= 0 TO 15 DO
	FOR nIdxAdr:= 0 TO 63 DO
		IF GVL_DALI.g_arrAddrInGroups[DALI_LINE_NUM].arrAddrInGroups[nIdxAdr, nIdxGrp] THEN
			GVL_DALI.g_arrAddrInGroups[DALI_LINE_NUM].arrAddressesInEachGroup[nIdxGrp, arrIDXCount[nIdxGrp] ]:= nIdxAdr ;
			arrIDXCount[nIdxGrp] := arrIDXCount[nIdxGrp] +1;
		END_IF
	END_FOR
END_FOR
END_ACTION

{attribute 'monitoring' := 'call'}
PROPERTY ipDALICommunication : Tc3_DALI.I_DALICommunication
GET
ipDALICommunication := THIS^.ipCommunication;
END_GET
SET
THIS^.ipCommunicationPreset := ipDALICommunication;
END_SET
END_PROPERTY

//| Apply the perset value of IpCommunication if available
//| Return codes:
//|   FALSE: no peset value available
//|   TRUE: has taken the preset value
{attribute 'hide'}
METHOD PRIVATE TrySetCommunication : BOOL
VAR_INPUT
END_VAR
IF ((THIS^.ipCommunication <> THIS^.ipCommunicationPreset) AND (THIS^.ipCommunicationPreset <> 0)) THEN
	THIS^.ipCommunication := THIS^.ipCommunicationPreset;
	THIS^.fbDALI102QueryStatus.ipDALICommunication := THIS^.ipCommunication;
	THIS^.fbDALI102QueryGroups.ipDALICommunication := THIS^.ipCommunication;
	THIS^.fbDALI102QueryLampFailure.ipDALICommunication := THIS^.ipCommunication;
	THIS^.fbDALI102Addressing.ipDALICommunication := THIS^.ipCommunication;
	THIS^.fbDALI102AddToGroup.ipDALICommunication := THIS^.ipCommunication;
	THIS^.fbDALI102QueryMissingShortAddress.ipDALICommunication := THIS^.ipCommunication;
	TrySetCommunication := TRUE;
ELSE
	TrySetCommunication := FALSE;
END_IF
END_METHOD

END_FUNCTION_BLOCK

// POUs/DALI/Ballast/FB_DALI_EnergyDataManagement
FUNCTION_BLOCK FB_DALI_EnergyDataManagement
(*
EnergyReporting reads ActiveEnergy (part 252) for all present ballasts on all (configured) DALI-lines where GVL_DALI.g_arrEnergyData[*DALI-line*,*ballast*].bHasEnergyData is TRUE.
Results are stored in GVL_DALI.g_arrEnergyData[*DALI-line*,*ballast*].fActiveEnergy. Energy Data for individual ballasts is NOT persistent in PLC, since the values are stored in the gear driver.
The engergy sum per DALI-Line (Wh) and Total Energy (Wh) are persistent.

If bCheckActiveEnergy is TRUE, all present ballasts are queried for ActiveEnergy and bHasEnergyData is updated accordingly.
This will result in errors for any ballast that does not comply with part 252. 
Errors will not be triggered for activations where bCheckActiveEnergy is FALSE.
Some values stored in gear drivers with major firmware version 96 are dubious. Max trust values are implemented.

During restart of PLC following an uninteded shutdown or download , EnergyReporting is activated automatically internally with bCheckActiveEnergy set to TRUE

EnergyReporting is activated automatically at TOD 0:00, 6:00, 12:00, 18:00 GMT (configurable) from the AHx_y program.

NB:	The priority of commands are set to "middle" internally. Updating all lines will take a couple of minutes to finish, so be patient.
	Other critical commands on the DALI-lines take priotity.
	Add appropriate communication immediately after configuration of a new KL6821 terminal in the AHx_y program.
	That is, arrfbDALI_EnergyReporting[*DALI-Line*].ipDALICommunication := P_DALI_Background.arrfbKL6821Communication[*DALI-Line*];
*)
VAR_INPUT
	
	NumOfEnergyLines				: BYTE;
END_VAR
VAR_IN_OUT
	bReadEnergyDataAllLines			: BOOL;
	arrfbDALI_EnergyReporting		: ARRAY[1..DALI_Param.MAX_DALIV2_LINES] OF FB_DALI_EnergyReporting;
	arrDaliLineEnergySum			: ARRAY[1..DALI_Param.MAX_DALIV2_LINES] OF LREAL;
	fTotalEnergyWH					: LREAL;
	nMaxControlGearOperatingHours	: UINT;	
END_VAR

VAR_OUTPUT
	bReportingDone					: BOOL := FALSE;
	bErr							: BOOL;
END_VAR
VAR
	fbReadAllRTrig						: R_TRIG;
	arrReadEnergyData				: ARRAY[1..DALI_Param.MAX_DALIV2_LINES] OF BOOL;
	arrCheckActiveEnergy			: ARRAY[1..DALI_Param.MAX_DALIV2_LINES] OF BOOL;
	arrDone									: ARRAY[1..DALI_Param.MAX_DALIV2_LINES] OF BOOL;
	arrErr									: ARRAY[1..DALI_Param.MAX_DALIV2_LINES] OF BOOL;
	arrBusy									: ARRAY[1..DALI_Param.MAX_DALIV2_LINES] OF BOOL;
	arrContinue							: ARRAY[1..DALI_Param.MAX_DALIV2_LINES] OF BOOL;
	arrfbRTrigDone						: ARRAY[1..DALI_Param.MAX_DALIV2_LINES] OF R_TRIG;
	arrRTrigDone						: ARRAY[1..DALI_Param.MAX_DALIV2_LINES] OF BOOL;
	bContinueTest						: BOOL := TRUE;
	bCltsEveryContinueBool		: BOOL := FALSE;
	nFirstNotContinue					: DINT;
	fbRtrig_ReportingDone			: R_TRIG;
	byEnergyLineIdx 					: BYTE;
	
	//variables to store persistent data correctly
	byCount								: BYTE;
	arrMaxControlGearOperatingTimeTmp	: ARRAY[1..DALI_Param.MAX_DALIV2_LINES] OF UDINT;
	arrMaxControlGearOperatingTime		: ARRAY[1..DALI_Param.MAX_DALIV2_LINES] OF UDINT;
	nMaxControlGearOperatingHoursTmp	: UINT;
	//byShrtAddrOfMostUsedBallast		: ARRAY[1..DALI_Param.MAX_DALIV2_LINES] OF BYTE;
	arrDaliLineEnergySumTmp				: ARRAY[1..DALI_Param.MAX_DALIV2_LINES] OF LREAL;
	arrDaliLineEnergySumOld				: ARRAY[1..DALI_Param.MAX_DALIV2_LINES] OF LREAL;
	arrDaliLineEnergyChange				: ARRAY[1..DALI_Param.MAX_DALIV2_LINES] OF LREAL;
	fTotalEnergyChangeWHTmp				: LREAL;
	fMaxEnergyValueTrust				: LREAL := 1000000000;
	nMaxTimeValueTrust					: UDINT := 100000000;
	
END_VAR

(*
Program is a nested for loop from 1 to 63 in a for loop from 1 to MAX_DALIV2_LINES.
The nested loops do NOT wait for EnergyReporting to finish. The loops are entered only, when EnergyData has finished and data is available
*)
FOR byEnergyLineIdx := 1 TO DALI_Param.MAX_DALIV2_LINES DO
	IF bReadEnergyDataAllLines = TRUE THEN
		IF byEnergyLineIdx <= NumOfEnergyLines THEN			//Only read existing DALI lines
			arrReadEnergyData[byEnergyLineIdx] := TRUE;
		ELSE
			arrReadEnergyData[byEnergyLineIdx] := FALSE;
		END_IF
	END_IF;
	
	arrfbDALI_EnergyReporting[byEnergyLineIdx](
		bExecute:= arrReadEnergyData[byEnergyLineIdx], 
		DALI_LINE_NUM:= byEnergyLineIdx,
		bCheckActiveEnergy := arrCheckActiveEnergy[byEnergyLineIdx],
		bBusy=> arrBusy[byEnergyLineIdx], 
		bActionBusy=> , 
		bErr=> arrErr[byEnergyLineIdx], 
		nErrorId=> ,
		bDone =>  arrDone[byEnergyLineIdx]);
		
	arrContinue[byEnergyLineIdx] :=  arrDone[byEnergyLineIdx] OR arrErr[byEnergyLineIdx] AND NOT arrBusy[byEnergyLineIdx]; //If energy reporting for a line results in error, program still needs to finish
	
	arrfbRTrigDone[byEnergyLineIdx](CLK := arrDone[byEnergyLineIdx], Q => arrRTrigDone[byEnergyLineIdx]);
	IF arrRTrigDone[byEnergyLineIdx] THEN				//The moment a line is updated, EnergyReporting is deactivated, values are summed and max operating time found
		arrReadEnergyData[byEnergyLineIdx] := FALSE;
		bReadEnergyDataAllLines := FALSE;
		FOR byCount := 0 TO 63 DO
			IF GVL_DALI.g_arrEnergyData[byEnergyLineIdx, byCount].fActiveEnergy < fMaxEnergyValueTrust THEN				//Checking for dubious values
			arrDaliLineEnergySumTmp[byEnergyLineIdx] := arrDaliLineEnergySumTmp[byEnergyLineIdx] + GVL_DALI.g_arrEnergyData[byEnergyLineIdx, byCount].fActiveEnergy;
			END_IF
			IF GVL_DALI.g_arrEnergyData[byEnergyLineIdx, byCount].nControlGearOperatingTime < nMaxTimeValueTrust THEN				//Checking for dubious values
			arrMaxControlGearOperatingTimeTmp[byEnergyLineIdx] := MAX(arrMaxControlGearOperatingTimeTmp[byEnergyLineIdx], GVL_DALI.g_arrEnergyData[byEnergyLineIdx, byCount].nControlGearOperatingTime);
			END_IF
			IF byCount = 63 THEN			//The moment energy for a line is summed, the the sum is added to the total. Maximum operating time for the line is compared to current maximum
				arrDaliLineEnergySumOld[byEnergyLineIdx] := arrDaliLineEnergySum[byEnergyLineIdx];
				arrDaliLineEnergySum[byEnergyLineIdx] := arrDaliLineEnergySumTmp[byEnergyLineIdx];
				arrDaliLineEnergyChange[byEnergyLineIdx] := arrDaliLineEnergySum[byEnergyLineIdx] - arrDaliLineEnergySumOld[byEnergyLineIdx];
				IF arrDaliLineEnergyChange[byEnergyLineIdx] < 0 THEN
					arrDaliLineEnergyChange[byEnergyLineIdx] := 0;					//Only positive values allowed
				END_IF
				fTotalEnergyChangeWHTmp := fTotalEnergyChangeWHTmp + arrDaliLineEnergyChange[byEnergyLineIdx];
				arrDaliLineEnergySumTmp[byEnergyLineIdx] := 0;
				arrMaxControlGearOperatingTime[byEnergyLineIdx] := arrMaxControlGearOperatingTimeTmp[byEnergyLineIdx];
				arrMaxControlGearOperatingTimeTmp[byEnergyLineIdx] := 0;
				nMaxControlGearOperatingHoursTmp := MAX(nMaxControlGearOperatingHoursTmp, TO_UINT(TRUNC(arrMaxControlGearOperatingTime[byEnergyLineIdx]*EXPT(60,-2)))); //Maximum is converted to REAL and hours - then converted to UINT. Maximum of positive numbers are positive. As so the conversion to UINT is appropriate. 
			END_IF
		END_FOR
	END_IF
END_FOR

//Checking if configured DALI-lines are done or resulted in error but not busy
bCltsEveryContinueBool := F_CltsEveryBool(
	bTest			:= bContinueTest,
	in				:= arrContinue,
	index			=> nFirstNotContinue		
	);
fbReadAllRTrig(CLK:=bReadEnergyDataAllLines);
IF (NumOfEnergyLines < nFirstNotContinue OR bCltsEveryContinueBool) AND NOT fbReadAllRTrig.Q THEN
	bReportingDone := TRUE;
ELSE
	bReportingDone := FALSE;
END_IF

//The moment the total is calculated and maximum found the values are returned and temp values are reset
fbRtrig_ReportingDone(CLK:=bReportingDone);
IF fbRtrig_ReportingDone.Q AND NOT fbReadAllRTrig.Q THEN 
		nMaxControlGearOperatingHours := nMaxControlGearOperatingHoursTmp;
		nMaxControlGearOperatingHoursTmp := 0;
		fTotalEnergyWH := fTotalEnergyWH + fTotalEnergyChangeWHTmp;
		fTotalEnergyChangeWHTmp := 0;
		bReadEnergyDataAllLines := FALSE;
END_IF

END_FUNCTION_BLOCK

// POUs/Misc/F_CltsEveryBool
FUNCTION F_CltsEveryBool : BOOL

VAR_INPUT

    bTest: BOOL;

END_VAR

VAR_IN_OUT

    in: ARRAY[*] OF BOOL;

END_VAR

VAR_OUTPUT

    index: DINT;

END_VAR

VAR

                i: DINT;

END_VAR

F_CltsEveryBool := TRUE;   // Assume success by default

index := -1;             // Default index when all match

 

FOR i := LOWER_BOUND(in, 1) TO UPPER_BOUND(in, 1) DO

    IF in[i] <> bTest THEN

        F_CltsEveryBool := FALSE; // Found a mismatch

        index := i;             // Report failing index

        EXIT;                 // Exit early

    END_IF

END_FOR

END_FUNCTION

// POUs/DALI/Ballast/FB_DALI_EnergyReporting
FUNCTION_BLOCK FB_DALI_EnergyReporting
VAR_INPUT
	bExecute							: BOOL;
	DALI_LINE_NUM						: BYTE;	(*DALI-Linie//DALI-line*)
END_VAR
VAR_IN_OUT
bCheckActiveEnergy						: BOOL;
END_VAR
VAR_OUTPUT
	bBusy								: BOOL;
	bActionBusy 						: BOOL;
	bErr								: BOOL;	
	nErrorId							: UDINT;
	bDone								: BOOL;
END_VAR
VAR
	ipCommunication							: I_DALICommunication;
	ipCommunicationPreset					: I_DALICommunication;

	fbDALI252QueryActiveEnergy				: FB_DALI252QueryActiveEnergy(0);
	fbDALI252QueryActiveEnergyLoadside		: FB_DALI252QueryActiveEnergyLoadside(0);
	fbDALI252QueryActivePower				: FB_DALI252QueryActivePower(0);
	fbDALI252QueryActivePowerLoadside 		: FB_DALI252QueryActivePowerLoadside(0);
	fbDALI252QueryApparentEnergy 			: FB_DALI252QueryApparentEnergy(0);
	fbDALI252QueryApparentPower 			: FB_DALI252QueryApparentPower(0);
	
	fbDALI253QueryControlGearOperatingTime 	: FB_DALI253QueryControlGearOperatingTime(0);
	fbDALI253QueryControlGearStartCounter 	: FB_DALI253QueryControlGearStartCounter(0);
	fbDALI253QueryLightSourceStartCounter 	: FB_DALI253QueryLightSourceStartCounter(0);
	
	
	bInit									: BOOL;
	byShrtAdr								: BYTE:=1;	

	byCount									: BYTE;
	uiCmdStep								: INT;
	bCallData								: BOOL;
	
	fbRTrigInitDevice						: R_TRIG;

	bInitReadEnergyOK: BOOL;
END_VAR

{region "initialize the outputs"}
IF (NOT bInit) THEN
	THIS^.TrySetCommunication();		 
	bBusy := TRUE;
	nErrorId := 0;
	bErr := FALSE;
	bInit := TRUE;
END_IF
{endregion}

{region "check parameters"}
IF (ipCommunication = 0) THEN
	bErr := TRUE;
	nErrorId := TC_EVENTS.TcDALIEventClass.TheInterfaceToTheCommunicationBufferIsNotInitialized.nEventId;
	uiCmdStep := 0;
END_IF

IF (byShrtAdr > 63) THEN
	bErr := TRUE;
	nErrorId := 16#8000; // custom error code: Parameter byShrtAdr lies outside of the valid range
	uiCmdStep := 0;		 
END_IF
{endregion}

fbRTrigInitDevice(CLK:= GVL_DALI.g_arrDiagnosisRunOnce[DALI_LINE_NUM] , Q=> );
IF fbRTrigInitDevice.Q THEN
	bCheckActiveEnergy := TRUE;
END_IF
IF fbRTrigInitDevice.Q THEN
	bCallData:= TRUE;
	bDone := FALSE;
END_IF
IF GVL_DALI.g_arrDiagnosisRunOnce[DALI_LINE_NUM] AND bExecute THEN
	bCallData:= TRUE;
	bDone := FALSE;
END_IF

IF NOT (bBusy OR bDone) THEN
	IF bCallData THEN
		bBusy := TRUE;
		A_ResetRoutine();
		byCount := 0;
		uiCmdStep:=10;
	END_IF	
END_IF


CASE uiCmdStep OF

0: (*Idle*)
	bBusy := FALSE;
	bCallData:= FALSE;
	
10:
	IF bCallData = TRUE THEN 
		arrbBlockDTR[DALI_LINE_NUM] := TRUE;
		IF GVL_DALI.g_arrGrpAssignment[DALI_LINE_NUM, byCount].bLampPresentInNetwork AND (bCheckActiveEnergy OR g_arrEnergyData[DALI_LINE_NUM, byCount].bHasEnergyData) THEN
			byShrtAdr := byCount;
			uiCmdStep := 100;
			
		ELSE
			uiCmdStep := 11;
		END_IF
	END_IF
		
11:
	IF byCount >= 63 THEN
		byCount:= 0 ;
		uiCmdStep:= 0;
		arrbBlockDTR[DALI_LINE_NUM]:=FALSE;
		bDone := TRUE;
		bCheckActiveEnergy := FALSE;
	ELSE
		byCount:= byCount + 1;
		uiCmdStep := 10;
	END_IF
	
100: //Reset and make sure we are ready for new commands
	A_ResetRoutine();
	IF NOT bActionBusy	THEN
		IF bErr	THEN
			uiCmdStep:= 0;
			arrbBlockDTR[DALI_LINE_NUM]:=FALSE;
		ELSE
			uiCmdStep:= 101;
		END_IF
	END_IF

101:(*Query Active Energy*)
	A_DALI252QueryActiveEnergy();
	IF NOT bActionBusy	THEN
		IF bErr	THEN
			uiCmdStep:= 11;
			arrbBlockDTR[DALI_LINE_NUM]:=FALSE;
		ELSE
			uiCmdStep:= 120; //Skip to the data we need
		END_IF
	END_IF
	
110:
	IF NOT bActionBusy	THEN
		IF bErr	THEN
			uiCmdStep:= 0;
			arrbBlockDTR[DALI_LINE_NUM]:=FALSE;
		ELSE
			uiCmdStep:= 111;
		END_IF
	END_IF

111:(*Query Active Energy*)
	A_DALI252QueryActiveEnergyLoadside();
	IF NOT bActionBusy	THEN
		IF bErr	THEN
			uiCmdStep:= 0;
			arrbBlockDTR[DALI_LINE_NUM]:=FALSE;
		ELSE
			uiCmdStep:= 120;
		END_IF
	END_IF
		
120:
	IF NOT bActionBusy	THEN
		IF bErr	THEN
			uiCmdStep:= 0;
			arrbBlockDTR[DALI_LINE_NUM]:=FALSE;
		ELSE
			uiCmdStep:= 121;
		END_IF
	END_IF

121:(*Query Active Power*)
	A_DALI252QueryActivePower();
	IF NOT bActionBusy	THEN
		IF bErr	THEN
			uiCmdStep:= 0;
			arrbBlockDTR[DALI_LINE_NUM]:=FALSE;
		ELSE
			uiCmdStep:= 160; //Skip to the data we need
		END_IF
	END_IF

130:
	IF NOT bActionBusy	THEN
		IF bErr	THEN
			uiCmdStep:= 0;
			arrbBlockDTR[DALI_LINE_NUM]:=FALSE;
		ELSE
			uiCmdStep:= 131;
		END_IF
	END_IF

131:(*Query Active Energy*)
	A_DALI252QueryActiveEnergyLoadside();
	IF NOT bActionBusy	THEN
		IF bErr	THEN
			uiCmdStep:= 0;
			arrbBlockDTR[DALI_LINE_NUM]:=FALSE;
		ELSE
			uiCmdStep:= 140;
		END_IF
	END_IF

140:
	IF NOT bActionBusy	THEN
		IF bErr	THEN
			uiCmdStep:= 0;
			arrbBlockDTR[DALI_LINE_NUM]:=FALSE;
		ELSE
			uiCmdStep:= 141;
		END_IF
	END_IF

141:(*Query Active Energy*)
	A_DALI252QueryApparentPower();
	IF NOT bActionBusy	THEN
		IF bErr	THEN
			uiCmdStep:= 0;
			arrbBlockDTR[DALI_LINE_NUM]:=FALSE;
		ELSE
			uiCmdStep:= 150;
		END_IF
	END_IF

150:
	IF NOT bActionBusy	THEN
		IF bErr	THEN
			uiCmdStep:= 0;
			arrbBlockDTR[DALI_LINE_NUM]:=FALSE;
		ELSE
			uiCmdStep:= 151;
		END_IF
	END_IF

151:(*Query Active Energy*)
	A_DALI252QueryApparentEnergy();
	IF NOT bActionBusy	THEN
		IF bErr	THEN
			uiCmdStep:= 0;
			arrbBlockDTR[DALI_LINE_NUM]:=FALSE;
		ELSE
			uiCmdStep:= 160;
		END_IF
	END_IF	

160:
	IF NOT bActionBusy	THEN
		IF bErr	THEN
			uiCmdStep:= 0;
			arrbBlockDTR[DALI_LINE_NUM]:=FALSE;
		ELSE
			uiCmdStep:= 161;
		END_IF
	END_IF

161:(*Query Active Energy*)
	A_DALI253QueryControlGearOperatingTime();
	IF NOT bActionBusy	THEN
		IF bErr	THEN
			uiCmdStep:= 0;
			arrbBlockDTR[DALI_LINE_NUM]:=FALSE;
		ELSE
			uiCmdStep:= 888;
		END_IF
	END_IF		
	
888: //Done step
	IF byCount>=63 THEN
		uiCmdStep:=0;
		byCount := 0;
		bInitReadEnergyOK := TRUE;
		arrbBlockDTR[DALI_LINE_NUM]:=FALSE;
		bCheckActiveEnergy := FALSE;
		bDone := TRUE;
	ELSE
		byCount:= byCount + 1;
		uiCmdStep:= 10;
	END_IF
	
END_CASE

ACTION A_DALI252QueryActiveEnergy:
bActionBusy	:= TRUE;
	

fbDALI252QueryActiveEnergy(
	bError=> , 
	ipResultMessage=> , 
	bStart:= TRUE , 
	nAddress:= byShrtAdr, 
	eAddressType:= E_DALIAddressType.Short, 
	eCommandPriority:= E_DALICommandPriority.Middle, 
	bBusy=>);
	

	IF NOT fbDALI252QueryActiveEnergy.bBusy	THEN
		IF	fbDALI252QueryActiveEnergy.bError	THEN
			bErr     	:= TRUE;
			nErrorId := fbDALI252QueryActiveEnergy.ipResultMessage.nEventId;
			GVL_DALI.g_arrEnergyData[DALI_LINE_NUM, byShrtAdr].bHasEnergyData := FALSE;
		ELSE GVL_DALI.g_arrEnergyData[DALI_LINE_NUM, byShrtAdr].bHasEnergyData := TRUE;
		END_IF
		bActionBusy		:= FALSE;
		GVL_DALI.g_arrEnergyData[DALI_LINE_NUM, byShrtAdr].fActiveEnergy:= ULINT_TO_REAL(fbDALI252QueryActiveEnergy.nActiveEnergy) * EXPT(10,fbDALI252QueryActiveEnergy.nScaleFactorForActiveEnergy);
		fbDALI252QueryActiveEnergy(bStart:= FALSE );
	END_IF
END_ACTION

ACTION A_DALI252QueryActiveEnergyLoadside:
bActionBusy	:= TRUE;
	

fbDALI252QueryActiveEnergyLoadside(
	bError=> , 
	ipResultMessage=> , 
	bStart:= TRUE , 
	nAddress:= byShrtAdr, 
	eAddressType:= E_DALIAddressType.Short, 
	eCommandPriority:= E_DALICommandPriority.Middle, 
	bBusy=> );
	

	IF NOT fbDALI252QueryActiveEnergyLoadside.bBusy	THEN
		IF	fbDALI252QueryActiveEnergyLoadside.bError	THEN
			bErr     	:= TRUE;
			nErrorId := fbDALI252QueryActiveEnergyLoadside.ipResultMessage.nEventId;
		END_IF
		bActionBusy		:= FALSE;
		GVL_DALI.g_arrEnergyData[DALI_LINE_NUM, byShrtAdr].fActiveEnergyLoadside:= ULINT_TO_REAL(fbDALI252QueryActiveEnergyLoadside.nActiveEnergyLoadside) * EXPT(10,fbDALI252QueryActiveEnergyLoadside.nScaleFactorForLoadsideEnergy); 
		fbDALI252QueryActiveEnergyLoadside(bStart:= FALSE );
	END_IF
END_ACTION

ACTION A_DALI252QueryActivePower:
bActionBusy	:= TRUE;
	

fbDALI252QueryActivePower(
	bError=> , 
	ipResultMessage=> , 
	bStart:= TRUE , 
	nAddress:= byShrtAdr, 
	eAddressType:= E_DALIAddressType.Short, 
	eCommandPriority:= E_DALICommandPriority.Middle, 
	bBusy=> );
	

	IF NOT fbDALI252QueryActivePower.bBusy	THEN
		IF	fbDALI252QueryActivePower.bError	THEN
			bErr     	:= TRUE;
			nErrorId := fbDALI252QueryActivePower.ipResultMessage.nEventId;
		END_IF
		bActionBusy		:= FALSE;
		GVL_DALI.g_arrEnergyData[DALI_LINE_NUM, byShrtAdr].fActivePower:= ULINT_TO_REAL(fbDALI252QueryActivePower.nActivePower) * EXPT(10,fbDALI252QueryActivePower.nScaleFactorForActivePower); 
		fbDALI252QueryActivePower(bStart:= FALSE );
	END_IF
END_ACTION

ACTION A_DALI252QueryActivePowerLoadside:
bActionBusy	:= TRUE;
	

fbDALI252QueryActivePowerLoadside(
	bError=> , 
	ipResultMessage=> , 
	bStart:= TRUE , 
	nAddress:= byShrtAdr, 
	eAddressType:= E_DALIAddressType.Short, 
	eCommandPriority:= E_DALICommandPriority.Middle, 
	bBusy=> );
	

	IF NOT fbDALI252QueryActivePowerLoadside.bBusy	THEN
		IF	fbDALI252QueryActivePowerLoadside.bError	THEN
			bErr     	:= TRUE;
			nErrorId := fbDALI252QueryActivePowerLoadside.ipResultMessage.nEventId;
		END_IF
		bActionBusy		:= FALSE;
		GVL_DALI.g_arrEnergyData[DALI_LINE_NUM, byShrtAdr].fActivePowerLoadside:= ULINT_TO_REAL(fbDALI252QueryActivePowerLoadside.nActivePowerLoadside) * EXPT(10,fbDALI252QueryActivePowerLoadside.nScaleFactorForLoadsidePower); 
		fbDALI252QueryActivePowerLoadside(bStart:= FALSE );
	END_IF
END_ACTION

ACTION A_DALI252QueryApparentEnergy:
bActionBusy	:= TRUE;
	

fbDALI252QueryApparentEnergy(
	bError=> , 
	ipResultMessage=> , 
	bStart:= TRUE , 
	nAddress:= byShrtAdr, 
	eAddressType:= E_DALIAddressType.Short, 
	eCommandPriority:= E_DALICommandPriority.Middle, 
	bBusy=>);
	

	IF NOT fbDALI252QueryApparentEnergy.bBusy	THEN
		IF	fbDALI252QueryApparentEnergy.bError	THEN
			bErr     	:= TRUE;
			nErrorId := fbDALI252QueryApparentEnergy.ipResultMessage.nEventId;
		END_IF
		bActionBusy		:= FALSE;
		GVL_DALI.g_arrEnergyData[DALI_LINE_NUM, byShrtAdr].fApparentEnergy:= ULINT_TO_REAL(fbDALI252QueryApparentEnergy.nApparentEnergy) * EXPT(10,fbDALI252QueryApparentEnergy.nScaleFactorForApparentEnergy); 
		fbDALI252QueryApparentEnergy(bStart:= FALSE );
	END_IF
END_ACTION

ACTION A_DALI252QueryApparentPower:
bActionBusy	:= TRUE;
	

fbDALI252QueryApparentPower(
	bError=> , 
	ipResultMessage=> , 
	bStart:= TRUE , 
	nAddress:= byShrtAdr, 
	eAddressType:= E_DALIAddressType.Short, 
	eCommandPriority:= E_DALICommandPriority.Middle, 
	bBusy=> );
	

	IF NOT fbDALI252QueryApparentPower.bBusy	THEN
		IF	fbDALI252QueryApparentPower.bError	THEN
			bErr     	:= TRUE;
			nErrorId := fbDALI252QueryApparentPower.ipResultMessage.nEventId;
		END_IF
		bActionBusy		:= FALSE;
		GVL_DALI.g_arrEnergyData[DALI_LINE_NUM, byShrtAdr].fApparentPower:= ULINT_TO_REAL(fbDALI252QueryApparentPower.nApparentPower) * EXPT(10,fbDALI252QueryApparentPower.nScaleFactorForApparentPower); 
		fbDALI252QueryApparentPower(bStart:= FALSE );
	END_IF
END_ACTION

ACTION A_DALI253QueryControlGearOperatingTime:
bActionBusy	:= TRUE;
	

fbDALI253QueryControlGearOperatingTime(
	bError=> , 
	ipResultMessage=> , 
	bStart:= TRUE , 
	nAddress:= byShrtAdr, 
	eAddressType:= E_DALIAddressType.Short, 
	eCommandPriority:= E_DALICommandPriority.Middle, 
	bBusy=> );
	

	IF NOT fbDALI253QueryControlGearOperatingTime.bBusy	THEN
		IF	fbDALI253QueryControlGearOperatingTime.bError	THEN
			bErr     	:= TRUE;
			nErrorId := fbDALI253QueryControlGearOperatingTime.ipResultMessage.nEventId;
		END_IF
		bActionBusy		:= FALSE;
		GVL_DALI.g_arrEnergyData[DALI_LINE_NUM, byShrtAdr].nControlGearOperatingTime:= fbDALI253QueryControlGearOperatingTime.nControlGearOperatingTime; 
		fbDALI253QueryControlGearOperatingTime(bStart:= FALSE );
	END_IF
END_ACTION

ACTION A_DALI253QueryControlGearStartCounter:
bActionBusy	:= TRUE;
	

fbDALI253QueryControlGearOperatingTime(
	bError=> , 
	ipResultMessage=> , 
	bStart:= TRUE , 
	nAddress:= byShrtAdr, 
	eAddressType:= E_DALIAddressType.Short, 
	eCommandPriority:= E_DALICommandPriority.Middle, 
	bBusy=> );
	

	IF NOT fbDALI253QueryControlGearStartCounter.bBusy	THEN
		IF	fbDALI253QueryControlGearStartCounter.bError	THEN
			bErr     	:= TRUE;
			nErrorId := fbDALI253QueryControlGearStartCounter.ipResultMessage.nEventId;
		END_IF
		bActionBusy		:= FALSE;
		GVL_DALI.g_arrEnergyData[DALI_LINE_NUM, byShrtAdr].nControlGearStartCounter:= fbDALI253QueryControlGearStartCounter.nControlGearStartCounter; 
		fbDALI253QueryControlGearStartCounter(bStart:= FALSE );
	END_IF
END_ACTION

ACTION A_DALI253QueryLightSourceStartCounter:
bActionBusy	:= TRUE;
	

fbDALI253QueryLightSourceStartCounter(
	bError=> , 
	ipResultMessage=> , 
	bStart:= TRUE , 
	nAddress:= byShrtAdr, 
	eAddressType:= E_DALIAddressType.Short, 
	eCommandPriority:= E_DALICommandPriority.Middle, 
	bBusy=> );
	

	IF NOT fbDALI253QueryLightSourceStartCounter.bBusy	THEN
		IF	fbDALI253QueryLightSourceStartCounter.bError	THEN
			bErr     	:= TRUE;
			nErrorId := fbDALI253QueryLightSourceStartCounter.ipResultMessage.nEventId;
		END_IF
		bActionBusy		:= FALSE;
		GVL_DALI.g_arrEnergyData[DALI_LINE_NUM, byShrtAdr].nLightSourceStartCounter:= fbDALI253QueryLightSourceStartCounter.nLightSourceStartCounter; 
		fbDALI253QueryLightSourceStartCounter(bStart:= FALSE );
	END_IF
END_ACTION

ACTION A_ResetRoutine:

	bErr     	:= FALSE;
	nErrorId 	:= 0;
//	byCount		:= 0;
	fbDALI252QueryActiveEnergy				(bStart:= FALSE );
	fbDALI252QueryActiveEnergyLoadside		(bStart:= FALSE );
	fbDALI252QueryActivePower				(bStart:= FALSE );
	fbDALI252QueryActivePowerLoadside		(bStart:= FALSE );
	fbDALI252QueryApparentEnergy			(bStart:= FALSE );
	fbDALI252QueryApparentPower				(bStart:= FALSE );
	fbDALI253QueryControlGearOperatingTime	(bStart:= FALSE );
	fbDALI253QueryControlGearStartCounter	(bStart:= FALSE );
	fbDALI253QueryLightSourceStartCounter	(bStart:= FALSE );
END_ACTION

{attribute 'monitoring' := 'call'}
PROPERTY ipDALICommunication : Tc3_DALI.I_DALICommunication
GET
ipDALICommunication := THIS^.ipCommunication;
END_GET
SET
THIS^.ipCommunicationPreset := ipDALICommunication;
END_SET
END_PROPERTY

//| Apply the perset value of IpCommunication if available
//| Return codes:
//|   FALSE: no peset value available
//|   TRUE: has taken the preset value
{attribute 'hide'}
METHOD PRIVATE TrySetCommunication : BOOL
VAR_INPUT
END_VAR
IF ((THIS^.ipCommunication <> THIS^.ipCommunicationPreset) AND (THIS^.ipCommunicationPreset <> 0)) THEN
	THIS^.ipCommunication := THIS^.ipCommunicationPreset;
	THIS^.fbDALI252QueryActiveEnergy.ipDALICommunication := THIS^.ipCommunication;
	THIS^.fbDALI252QueryActiveEnergyLoadside.ipDALICommunication := THIS^.ipCommunication;
	THIS^.fbDALI252QueryActivePower.ipDALICommunication := THIS^.ipCommunication;
	THIS^.fbDALI252QueryActivePowerLoadside.ipDALICommunication := THIS^.ipCommunication;
	THIS^.fbDALI252QueryApparentEnergy.ipDALICommunication := THIS^.ipCommunication;
	THIS^.fbDALI252QueryApparentPower.ipDALICommunication := THIS^.ipCommunication;
	THIS^.fbDALI253QueryControlGearOperatingTime.ipDALICommunication := THIS^.ipCommunication;
	THIS^.fbDALI253QueryControlGearStartCounter.ipDALICommunication := THIS^.ipCommunication;
	THIS^.fbDALI253QueryLightSourceStartCounter.ipDALICommunication := THIS^.ipCommunication;	
	TrySetCommunication := TRUE;
ELSE
	TrySetCommunication := FALSE;
END_IF
END_METHOD

END_FUNCTION_BLOCK

// POUs/DALI/Ballast/FB_DALILgtActr_EX
FUNCTION_BLOCK FB_DALILgtActr_EX  (* V1.1 dfgdfgdfgdfgdfgfzxcv *)
VAR_INPUT
	byShrtAdr				: BYTE;
	byGrpAdr				: BYTE;
	eMod					: E_DALIAddressType:= E_DALIAddressType.Group;
	fSttupCtrlVal			: REAL;
	fMinCtrlVal				: REAL;
	fMaxCtrlVal				: REAL;
	fLgtOffset				: REAL;
	eFadeTime				: E_DALIFadeTime:= E_DALIFadeTime.T02000ms;
	eFadeRate				: E_DALIFadeRate:= E_DALIFadeRate.N063StepsPerSec;
	uiBlinkTi				: UINT;
	uiOffDly				: UINT;
	uiPollActLgtLvl			: UINT;
	bReInit					: BOOL;
	nCycleTimeInMS			: UDINT;
	stLgtCmd				: ST_LgtCmd;
	DALI_LINE_NUM			: BYTE;
END_VAR
VAR_OUTPUT
	fActlLgtLvl				: REAL;
	byActlLgtLvl			: BYTE;
	bLgt					: BOOL;
	fActlMinCtrlVal			: REAL;
	bMinCtrlValRchd 		: BOOL;
	fActlMaxCtrlVal			: REAL;
	bMaxCtrlValRchd 		: BOOL;
	fRstVal					: REAL;
	eActlFadeTime			: E_DALIFadeTime;
	eActlFadeRate			: E_DALIFadeRate;
	byPhysMinVal			: BYTE;
	byActlMinCtrlVal		: BYTE;
	byActlMaxCtrlVal		: BYTE;
	bInitDevice				: BOOL;
	bBlinkSeqStarted 		: BOOL;
	bActionBusy				: BOOL;
	bErr     				: BOOL;
	nErrorId				: UDINT;
	byDALIDevSta			: BYTE;
END_VAR
VAR
	ipCommunication					: I_DALICommunication;
	ipCommunicationPreset			: I_DALICommunication;

	bInit					: BOOL;
	bBusy					: BOOL;
	bRstErr					: BOOL;
	rtReInit				: R_TRIG;
	bReactCmdSt				: BOOL;
	byAddr					: BYTE;
	eAddrType				: E_DALIAddressType;
	byArcPowerLevel			: BYTE;
	byDTR					: BYTE;
	uiCmdStep				: UINT;
	eFadeTime_SV			: E_DALIFadeTime;
	eFadeRate_SV			: E_DALIFadeRate;
	fMinCtrlVal_SV			: REAL;
	fMaxCtrlVal_SV			: REAL;
	bSetFadeRate			: BOOL;
	bSetFadeTime			: BOOL;
	bDimUp					: BOOL;
	bDimDwn					: BOOL;
	bySetFadeRate			: BYTE;
	bSetMinValInput			: BOOL;	(*Änderung MinVal über Bausteineingang*)
	bSetMaxValInput			: BOOL;	(*Änderung MaxVal über Bausteineingang*)
	bySetMinValInput		: BYTE;
	bySetMaxValInput		: BYTE;
	bSetMinValCmdSt			: BOOL;	(*Änderung MinVal über Kommandostruktur*)
	bSetMaxValCmdSt			: BOOL;	(*Änderung MaxVal über Kommandostruktur*)
	bySetMinValCmdSt		: BYTE;
	bySetMaxValCmdSt		: BYTE;
	byRstVal				: BYTE;
	bySttupCtrlVal			: BYTE;
	rtInitDevice			: R_TRIG;
	rtOff					: R_TRIG;
	rtClMinCtrlVal			: R_TRIG;
	rtClMaxCtrlVal			: R_TRIG;
	rtClOnVal				: R_TRIG;
	rtClRstVal				: R_TRIG;
	rtSetCtrlValDct			: R_TRIG;
	rtChgMaxCtrlVal			: R_TRIG;
	rtChgMinCtrlVal			: R_TRIG;
	rtStpUp							: R_TRIG;
	rtStpDwn						: R_TRIG;
	rtRmp							: R_TRIG;
	tonSeqTimer						: TON;
	tonDimRepeat					: TON;
	fbUp							: FB_DALI102Up(0);
	fbDwn							: FB_DALI102Down(0);
	fbOff							: FB_DALI102Off(0);
	fbRecallMaxLevel				: FB_DALI102RecallMaxLevel(0);
	fbRecallMinLevel				: FB_DALI102RecallMinLevel(0);
	fbDirectArcPowerControl			: FB_DALI102DirectArcPowerControl(0);
	fbStepUp						: FB_DALI102StepUp(0);
	fbStepDown						: FB_DALI102StepDown(0);
	fbQueryActualLevel				: FB_DALI102QueryActualLevel(0);
	fbSetFadeRate					: FB_DALI102SetFadeRate(0);
	fbSetFadeTime					: FB_DALI102SetFadeTime(0);
	fbSetMinLevel					: FB_DALI102SetMinLevel(0);
	fbQueryMinLevel					: FB_DALI102QueryMinLevel(0);
	fbQueryMaxLevel					: FB_DALI102QueryMaxLevel(0);
	fbQueryPhysicalMinLevel			: FB_DALI102QueryPhysicalMinimum(0);
	fbSetMaxLevel					: FB_DALI102SetMaxLevel(0);
	fbQueryActualLevelBackgound		: FB_DALI102QueryActualLevel(0);
	fbQueryStatusBackground			: FB_DALI102QueryStatus(0);
	fbSendValue						: FB_BA_ValTrigf;
	fbReTrigSend0					: R_TRIG;
	nStepQueryActualLevel			: UINT;
	tonCycleActualLevelMasterDev	: TON;
	bSetRetry						: BOOL;
	fbTimeOut						: TON;
	byActlFadeTime					: BYTE;
	nCycleCountSP					: UDINT;
	nActualCount					: UDINT:= 1;
	bInitDone: BOOL;
	bInitCom: BOOL;
END_VAR
VAR_IN_OUT
END_VAR


(* For checking which task the FB are called*)
IF nCycleTimeInMS > 0 THEN	(*nCycleCountSP are only calculated if nCycleTimeInMS are larger than 0*)
	nCycleCountSP:= (200 / nCycleTimeInMS) ; (* 200 are the target time between 2 UP/Down cmd*)
END_IF

{region "initialize the outputs"}
IF (NOT bInitCom) THEN
	THIS^.TrySetCommunication();		 
	bBusy := TRUE;
	nErrorId := 0;
	bErr := FALSE;
	bInitCom := TRUE;
	bInitDone := FALSE;
END_IF
{endregion}


{region "check parameters"}
IF (ipCommunication = 0) THEN
	bErr := TRUE;
	nErrorId := TC_EVENTS.TcDALIEventClass.TheInterfaceToTheCommunicationBufferIsNotInitialized.nEventId;
	uiCmdStep := 0;
END_IF
IF ((eMod <> E_DALIAddressType.Short) AND (eMod <> E_DALIAddressType.Group) AND (eMod <> E_DALIAddressType.Broadcast) AND (eMod <> E_DALIAddressType.BroadcastUnaddr)) THEN
	bErr := TRUE;
	nErrorId := TC_EVENTS.TcDALIEventClass.ParameterAddressTypeLiesOutsideOfTheValidRange.nEventId;
	uiCmdStep := 0;
END_IF
IF ((eMod = E_DALIAddressType.Short) AND (byShrtAdr > 63)) THEN
	bErr := TRUE;
	nErrorId := TC_EVENTS.TcDALIEventClass.ParameterAddressIsAShortAddressAndLiesOutsideOfTheValidRange.nEventId;
	uiCmdStep := 0;
END_IF
IF ((eMod = E_DALIAddressType.Group) AND (byGrpAdr > 15)) THEN
	bErr := TRUE;
	nErrorId := TC_EVENTS.TcDALIEventClass.ParameterAddressIsAGroupAddressAndLiesOutsideOfTheValidRange.nEventId;
	uiCmdStep := 0;
END_IF
IF (byShrtAdr > 63) THEN
	bErr := TRUE;
	nErrorId := 16#8000; // custom error code: Parameter byShrtAdr lies outside of the valid range
	uiCmdStep := 0;
END_IF
	
IF (byGrpAdr > 15) THEN
	bErr := TRUE;
	nErrorId := 16#8001; // custom error code: Parameter byGrpAdr lies outside of the valid range
	uiCmdStep := 0;
END_IF
{endregion}

(*	bRstErr ist ein Fehlermerker: wenn vorher über Fehler, s.o. herausgesprungen wurde und nun "alles gut" ist,
dann hier Fehler einmalig zurücksetzen, damit im weiteren Verlauf die Warnmeldungen sichtbar werden können*)
IF	bRstErr  THEN
		bRstErr    	:= FALSE;
		bErr     	:= FALSE;
END_IF


(* + + + + + + + + + + + + + + + + + + + + + + + + + + + + + + + + + + + + + + + + + + + + *)
(*In den DALI-Ausführungsaktionen ist jedoch zur Sicherheit noch ein RETURN-Aussprung*)
IF (eMod=E_DALIAddressType.Short)	THEN
	bReactCmdSt:=FALSE;
ELSE
	bReactCmdSt:=TRUE;
END_IF

(* + + + + + + + + + + + + + + + + + + + + + + + + + + + + + + + + + + + + + + + + + + + + *)
(*Init *)
rtReInit	 (CLK:=bReInit);
IF bReInit	THEN
	bInitDone:=FALSE;
END_IF

IF NOT bInitDone THEN
	rtInitDevice(CLK:=FALSE);
	bInitDevice				:= TRUE;
	fMinCtrlVal_SV			:= fMinCtrlVal;
	fMaxCtrlVal_SV			:= fMaxCtrlVal;
	bInit					:= TRUE;
	tonDimRepeat(PT:=T#200MS);

	IF fSttupCtrlVal < 0.0	 THEN
		bySttupCtrlVal	:= 0;
	ELSIF	fSttupCtrlVal > 100.0	 THEN
		bySttupCtrlVal	:= 254;
	ELSE
		bySttupCtrlVal	:= LREAL_TO_BYTE(F_fDALICurve(fSttupCtrlVal));
	END_IF
END_IF

rtInitDevice (CLK:=bInitDevice);

(* + + + + + + + + + + + + + + + + + + + + + + + + + + + + + + + + + + + + + + + + + + + + *)
(*Change DimTime/FadeRate über Bausteineingang*)
IF	(eFadeTime<>eFadeTime_SV) OR rtInitDevice.Q THEN
	eFadeTime_SV	:= eFadeTime;
	IF NOT rtInitDevice.Q	THEN
		bSetFadeRate	:= TRUE;
	END_IF
END_IF

IF	(eFadeRate<>eFadeRate_SV) OR rtInitDevice.Q THEN
	eFadeRate_SV	:= eFadeRAte;
	IF NOT rtInitDevice.Q	THEN
		bSetFadeRate	:= TRUE;
	END_IF
END_IF

(* + + + + + + + + + + + + + + + + + + + + + + + + + + + + + + + + + + + + + + + + + + + + *)
(*Change Min-/MaxCtrlVal über Bausteineingang*)

IF	(fMinCtrlVal<>fMinCtrlVal_SV) OR rtInitDevice.Q THEN
	fMinCtrlVal_SV		:= fMinCtrlVal;
	IF 		fMinCtrlVal < 0.0		 THEN
		bySetMinValInput	:= 0;
	ELSIF	fMinCtrlVal > 100.0	 THEN
		bySetMinValInput	:= 254;
	ELSE
		bySetMinValInput := LIMIT(0,LREAL_TO_BYTE(F_fDALICurve(fMinCtrlVal)), 254);
	END_IF
	IF NOT rtInitDevice.Q	THEN
		bSetMinValInput	:= TRUE;
	END_IF
END_IF

IF	(fMaxCtrlVal<>fMaxCtrlVal_SV) OR rtInitDevice.Q THEN
	fMaxCtrlVal_SV		:= fMaxCtrlVal;
	IF 		fMaxCtrlVal < 0.0		 THEN
		bySetMaxValInput	:= 0;
	ELSIF	fMaxCtrlVal > 100.0	 THEN
		bySetMaxValInput	:= 254;
	ELSE
		bySetMaxValInput := LIMIT(0,LREAL_TO_BYTE(F_fDALICurve(fMaxCtrlVal)), 254);

	END_IF
	IF NOT rtInitDevice.Q	THEN
		bSetMaxValInput	:= TRUE;
	END_IF
END_IF


(* + + + + + + + + + + + + + + + + + + + + + + + + + + + + + + + + + + + + + + + + + + + + *)
(*Change Min-/MaxCtrlVal über Kommandostruktur*)
rtChgMinCtrlVal	(CLK:= stLgtCmd.bChgMinCtrlVal);
rtChgMaxCtrlVal	(CLK:= stLgtCmd.bChgMaxCtrlVal);

IF 	rtChgMinCtrlVal.Q	AND bReactCmdSt			THEN
	IF 		stLgtCmd.fChgMinCtrlVal < 0.0		 THEN
		bySetMinValCmdSt	:= 0;
	ELSIF	stLgtCmd.fChgMinCtrlVal > 100.0	 THEN
		bySetMinValCmdSt	:= 254;
	ELSE
		bySetMinValCmdSt := LIMIT(0,LREAL_TO_BYTE(F_fDALICurve(stLgtCmd.fChgMinCtrlVal)), 254);
	END_IF
	bSetMinValCmdSt	:= TRUE;
END_IF

IF 	rtChgMaxCtrlVal.Q	AND bReactCmdSt			THEN
	IF 		stLgtCmd.fChgMaxCtrlVal < 0.0		 THEN
		bySetMaxValCmdSt	:= 0;
	ELSIF	stLgtCmd.fChgMaxCtrlVal > 100.0	 THEN
		bySetMaxValCmdSt	:= 254;
	ELSE
		bySetMaxValCmdSt := LIMIT(0,LREAL_TO_BYTE(F_fDALICurve(stLgtCmd.fChgMaxCtrlVal)), 254);
	END_IF
	bSetMaxValCmdSt	:= TRUE;
END_IF


fbSendValue(bEn:= TRUE, bRetrig:= , fIn:= stLgtCmd.fSetCtrlValDct, fHys:= 0.1);

IF bMinCtrlValRchd AND stLgtCmd.fSetCtrlValDct = 0 THEN
	fbReTrigSend0(CLK:=TRUE , Q=> );
ELSE
	fbReTrigSend0(CLK:=FALSE , Q=> );
END_IF

(* + + + + + + + + + + + + + + + + + + + + + + + + + + + + + + + + + + + + + + + + + + + + *)
(* Flankenbildung und Verriegelung der Schalt- und Dimmbefehle *)
rtOff			(CLK:=stLgtCmd.bOff OR fbReTrigSend0.Q);
rtClMinCtrlVal	(CLK:=stLgtCmd.bClMinCtrlVal);
rtClMaxCtrlVal	(CLK:=stLgtCmd.bClMaxCtrlVal);
rtClOnVal		(CLK:=stLgtCmd.bClOnVal);
rtClRstVal		(CLK:=stLgtCmd.bClRstVal);
rtSetCtrlValDct	(CLK:=stLgtCmd.bSetCtrlValDct OR fbSendValue.bSet);
rtStpUp			(CLK:=stLgtCmd.bStpUp);
rtStpDwn		(CLK:=stLgtCmd.bStpDwn);

bDimUp			:= stLgtCmd.bDimUp;
bDimDwn			:= stLgtCmd.bDimDwn;

(* + + + + + + + + + + + + + + + + + + + + + + + + + + + + + + + + + + + + + + + + + + + + *)
(* Prioritize of Commands *)
IF NOT bBusy	THEN
	IF			rtInitDevice.Q		THEN
				bBusy := TRUE;
				A_ResetRoutine();
				uiCmdStep:=1000;	
	ELSIF		bSetFadeRate	AND NOT bBlinkSeqStarted AND bInitDone THEN
				bBusy := TRUE;
				A_ResetRoutine();
				uiCmdStep:=300;
	ELSIF		bSetFadeTime	AND NOT bBlinkSeqStarted AND bInitDone THEN
				bBusy := TRUE;
				A_ResetRoutine();
				uiCmdStep:=305;
	ELSIF	bSetMinValInput		AND NOT bBlinkSeqStarted AND bInitDone THEN
				bBusy := TRUE;
				A_ResetRoutine();
				uiCmdStep:=310;
	ELSIF	bSetMaxValInput		AND NOT bBlinkSeqStarted AND bInitDone THEN
				bBusy := TRUE;
				A_ResetRoutine();
				uiCmdStep:=320;
	ELSIF	bSetMinValCmdSt		AND NOT bBlinkSeqStarted AND bInitDone THEN
				bBusy := TRUE;
				A_ResetRoutine();
				uiCmdStep:=330;
	ELSIF	bSetMaxValCmdSt		AND NOT bBlinkSeqStarted AND bInitDone THEN
				bBusy := TRUE;
				A_ResetRoutine();
				uiCmdStep:=340;
	ELSIF	bDimUp				AND NOT bMaxCtrlValRchd AND bInitDone THEN
				bBusy := TRUE;
				A_ResetRoutine();
				uiCmdStep:=10;
	ELSIF	bDimDwn				AND NOT bMinCtrlValRchd AND bInitDone THEN
				bBusy := TRUE;
				A_ResetRoutine();
				uiCmdStep:=20;
	ELSIF	rtOff.Q				AND bInitDone THEN
				bBusy := TRUE;
				A_ResetRoutine();
				uiCmdStep:=30;
	ELSIF	rtClMinCtrlVal.Q	AND bInitDone THEN
				bBusy := TRUE;
				A_ResetRoutine();
				uiCmdStep:=40;
	ELSIF	rtClMaxCtrlVal.Q	AND bInitDone THEN
				bBusy := TRUE;
				A_ResetRoutine();
				uiCmdStep:=50;
	ELSIF	rtClOnVal.Q	AND bInitDone THEN
				bBusy := TRUE;
				A_ResetRoutine();
				uiCmdStep:=60;
	ELSIF	rtClRstVal.Q		AND bInitDone THEN
				bBusy := TRUE;
				A_ResetRoutine();
				uiCmdStep:=70;
	ELSIF	rtSetCtrlValDct.Q	AND bInitDone THEN
				bBusy := TRUE;
				A_ResetRoutine();
				uiCmdStep:=80;
	ELSIF	rtStpUp.Q			AND NOT bMaxCtrlValRchd AND bInitDone THEN
				bBusy := TRUE;
				A_ResetRoutine();
				uiCmdStep:=90;
	ELSIF	rtStpDwn.Q			AND NOT bMinCtrlValRchd AND bInitDone THEN
				bBusy := TRUE;
				A_ResetRoutine();
				uiCmdStep:=100;
	END_IF
END_IF

(* + + + + + + + + + + + + + + + + + + + + + + + + + + + + + + + + + + + + + + + + + + + + *)
(*Kommandoausgabe*)
CASE uiCmdStep OF

0: (*Idle*)
	bInitDevice := FALSE;
	bBusy := FALSE;


(* - - - - - - - - - - - - - - - - - - - - - - - - *)
10:(*Dim Up*)
	bBlinkSeqStarted := FALSE;
(*	tonDimRepeat	(IN:=TRUE); *)  (*Disabled for at teste om Up cmd kommer hurtigere ved at tælle skan, istedet for timer*)
	nActualCount:= 1;
	A_DALICmdUp();
	IF NOT bActionBusy	THEN
		uiCmdStep:= 11;
	END_IF

11:(*Ende Wartezeit 200ms abwarten*)

(*Disablet to be more precise in case of long scantimes in the task - HMB 13/12-2021*)
(*	tonDimRepeat();
	IF tonDimRepeat.Q THEN
		tonDimRepeat(IN:= FALSE);
		IF bDimUp		THEN
			uiCmdStep:=10;
		ELSE
			uiCmdStep:=12;
		END_IF
	END_IF
*)
	(* Added to see if 200ms can be reached with this scan count*)
	IF nActualCount <= nCycleCountSP THEN
		nActualCount := nActualCount + 1;
		IF nActualCount >=nCycleCountSP THEN
			nActualCount:=1;
			IF bDimUp		THEN
				uiCmdStep:=10;
			ELSE
				uiCmdStep:=12;
			END_IF
		END_IF
	END_IF


12: (*Lichtabfrage wenn fertig*)
	A_DALICmdQueryActualLevel();
	IF NOT bActionBusy	THEN
		byActlLgtLvl	:= fbQueryActualLevel.nActualLevel;
		uiCmdStep		:= 0;
	END_IF

(* - - - - - - - - - - - - - - - - - - - - - - - - *)
20:(*Dim Down*)
	bBlinkSeqStarted := FALSE;
(*	tonDimRepeat	(IN:=TRUE); *)  (*Disabled for at teste om Up cmd kommer hurtigere ved at tælle skan, istedet for timer*)
	nActualCount:= 1;
	A_DALICmdDown();
	IF NOT bActionBusy	THEN
		uiCmdStep:= 21;
	END_IF

21:(*Ende Wartezeit 200ms abwarten*)
(*Disablet to be more precise in case of long scantimes in the task - HMB 13/12-2021*)
(*	tonDimRepeat();
	IF tonDimRepeat.Q THEN
		tonDimRepeat(IN:= FALSE);
		IF bDimDwn		THEN
			uiCmdStep:=20;
		ELSE
			uiCmdStep:=22;
		END_IF
	END_IF
*)
	IF nActualCount <= nCycleCountSP THEN
		nActualCount := nActualCount + 1;
		IF nActualCount >=nCycleCountSP THEN
			nActualCount:= 1;
			IF bDimDwn	THEN
				uiCmdStep:=20;
			ELSE
				uiCmdStep:=22;
			END_IF
		END_IF
	END_IF

22: (*Lichtabfrage wenn fertig*)
		A_DALICmdQueryActualLevel();
	IF NOT bActionBusy	THEN
		byActlLgtLvl	:= fbQueryActualLevel.nActualLevel;
		uiCmdStep		:= 0;
	END_IF

(* - - - - - - - - - - - - - - - - - - - - - - - - *)
30:(*Off*)
		A_DALICmdOff();
	IF NOT bActionBusy	THEN
		byActlLgtLvl	:=0;
		IF (uiOffDly<>0) AND NOT bBlinkSeqStarted AND NOT bErr	THEN
			uiCmdStep:=500;
		ELSE
			bBlinkSeqStarted := FALSE;
			uiCmdStep:= 0;
		END_IF
	END_IF

(* - - - - - - - - - - - - - - - - - - - - - - - - *)
40:(*Call MinCtrlVal*)
	bBlinkSeqStarted := FALSE;
	A_DALICmdRecallMinLevel();
	IF NOT bActionBusy	THEN
		byActlLgtLvl:=byActlMinCtrlVal;
		uiCmdStep:= 41;
	END_IF

41: (*Lichtabfrage wenn fertig*)
	A_DALICmdQueryActualLevel();
	IF NOT bActionBusy	THEN
		byActlLgtLvl	:= fbQueryActualLevel.nActualLevel;
		uiCmdStep		:= 0;
	END_IF	
	
(* - - - - - - - - - - - - - - - - - - - - - - - - *)
50:(*Call MaxCtrlVal*)
	bBlinkSeqStarted := FALSE;
		A_DALICmdRecallMaxLevel();
	IF NOT bActionBusy	THEN
		byActlLgtLvl:=byActlMaxCtrlVal;
		uiCmdStep:= 51;
	END_IF

51: (*Lichtabfrage wenn fertig*)
	A_DALICmdQueryActualLevel();
	IF NOT bActionBusy	THEN
		byActlLgtLvl	:= fbQueryActualLevel.nActualLevel;
		uiCmdStep		:= 0;
	END_IF	
	
(* - - - - - - - - - - - - - - - - - - - - - - - - *)
60:(*Call OnVal*)
	(*Limitation is not to be left to the electrical device -> the output of the actual value would be left to the background-polling only*)
	IF ((stLgtCmd.lrOnVal)>=fActlMaxCtrlVal)	THEN
		byArcPowerLevel:=byActlMaxCtrlVal;
	ELSIF ((stLgtCmd.lrOnVal)<=0.0)	THEN
		byArcPowerLevel:=0;
	ELSIF ((stLgtCmd.lrOnVal)<=fActlMinCtrlVal)	THEN
		byArcPowerLevel:=byActlMinCtrlVal;
	ELSE
		byArcPowerLevel := LIMIT(0,LREAL_TO_BYTE(F_fDALICurve(stLgtCmd.lrOnVal)), 254);
END_IF

		A_DALICmdDirectArcPowerControl();
	IF NOT bActionBusy	THEN
		byActlLgtLvl:=byRstVal;
		uiCmdStep:= 0;
	END_IF

(* - - - - - - - - - - - - - - - - - - - - - - - - *)
70:(*Call ResetVal*)
	bBlinkSeqStarted := FALSE;
	byArcPowerLevel	:= byRstVal;
		A_DALICmdDirectArcPowerControl();
	IF NOT bActionBusy	THEN
		byActlLgtLvl:=byRstVal;
		uiCmdStep:= 0;
	END_IF

(* - - - - - - - - - - - - - - - - - - - - - - - - *)
80:(*Set Control value directly*)
	(*Limitation is not to be left to the electrical device -> the output of the actual value would be left to the background-polling only*)
(*	IF (stLgtCmd.lrSetCtrlValDct+lrLgtOffset)>=lrActlMaxCtrlVal	THEN
		byArcPowerLevel:=byActlMaxCtrlVal;
	ELSIF (stLgtCmd.lrSetCtrlValDct+lrLgtOffset)<=0.0	THEN
		byArcPowerLevel:=0;
	ELSIF (stLgtCmd.lrSetCtrlValDct+lrLgtOffset)<=lrActlMinCtrlVal	THEN
		byArcPowerLevel:=byActlMinCtrlVal;
	ELSE

	END_IF
*)
	byArcPowerLevel:= LIMIT(0,LREAL_TO_BYTE(F_fDALICurve(stLgtCmd.fSetCtrlValDct + fLgtOffset)),254);
		A_DALICmdDirectArcPowerControl();
	IF NOT bActionBusy	THEN
(*		byActlLgtLvl:=byArcPowerLevel;*)
		IF (byActlLgtLvl=0) AND (uiOffDly<>0) AND NOT bBlinkSeqStarted AND NOT bErr	THEN
			uiCmdStep:=500;
		ELSE
			bBlinkSeqStarted := FALSE;
			IF stLgtCmd.bOff THEN
				uiCmdStep:= 0;
			ELSE
				uiCmdStep:= 0;
			END_IF
		END_IF	
	END_IF

81: (*Lichtabfrage wenn fertig*)
	A_DALICmdQueryActualLevel();
	IF NOT bActionBusy	THEN
		byActlLgtLvl	:= fbQueryActualLevel.nActualLevel;
		uiCmdStep		:= 0;
	END_IF	

(* - - - - - - - - - - - - - - - - - - - - - - - - *)
90:(*Step Up*)
	bBlinkSeqStarted := FALSE;
		A_DALICmdStepUp();
	IF NOT bActionBusy	THEN
		byActlLgtLvl:=byActlLgtLvl+1;
		IF	byActlLgtLvl>byActlMaxCtrlVal	THEN
			byActlLgtLvl:=byActlMaxCtrlVal;
		END_IF
		uiCmdStep:= 0;
	END_IF

(* - - - - - - - - - - - - - - - - - - - - - - - - *)
100:(*Step Down*)
	bBlinkSeqStarted := FALSE;
		A_DALICmdStepDown();
	IF NOT bActionBusy	THEN
		byActlLgtLvl:=byActlLgtLvl-1;
		IF	byActlLgtLvl<byActlMinCtrlVal	THEN
			byActlLgtLvl:=byActlMinCtrlVal;
		END_IF
		uiCmdStep:= 0;
	END_IF


(* - - - - - - - - - - - - - - - - - - - - - - - - *)
300:(*Set new FadeRate*)
	bSetFadeRate:=FALSE;
	IF NOT bActionBusy	THEN
		IF bErr	THEN
			uiCmdStep:= 0;
		ELSE
			uiCmdStep:= 301;
		END_IF
	END_IF

301:(*Set new FadeRate*)
	A_DALICmdSetFadeRate();
	IF NOT bActionBusy	THEN
		uiCmdStep:= 0;
	END_IF
	eActlFadeRate:=eFadeRate;
	
	
305:(*Set new FadeTime *)
	bSetFadeTime:=FALSE;
	IF NOT bActionBusy	THEN
		IF bErr	THEN
			uiCmdStep:= 0;
		ELSE
			uiCmdStep:= 306;
		END_IF
	END_IF

306:(*Set new FadeRate*)
	A_DALICmdSetFadeRate();
	IF NOT bActionBusy	THEN
		uiCmdStep:= 0;
	END_IF
	eActlFadeTime:=eFadeTime;

(* - - - - - - - - - - - - - - - - - - - - - - - - *)
310:(*Set new Min-Level*)
	bSetMinValInput:=FALSE;

	byDTR:=bySetMinValInput;
	IF NOT bActionBusy	THEN
		IF bErr	THEN
			uiCmdStep:= 0;
		ELSE
			uiCmdStep:= 311;
		END_IF
	END_IF

311:(*Set new MinLevel*)
		A_DALICmdSetMinLevel_Input();
	IF NOT bActionBusy	THEN
		IF bErr	THEN
			uiCmdStep:= 0;
		ELSE
			uiCmdStep:= 350;
		END_IF
	END_IF

(* - - - - - - - - - - - - - - - - - - - - - - - - *)
320:(*Set new MaxLevel *)
	bSetMaxValInput:=FALSE;

	byDTR:=bySetMaxValInput;
	IF NOT bActionBusy	THEN
		IF bErr	THEN
			uiCmdStep:= 0;
		ELSE
			uiCmdStep:= 321;
		END_IF
	END_IF

321:(*Set new MaxLevel*)
		A_DALICmdSetMaxLevel_Input();
	IF NOT bActionBusy	THEN
		IF bErr	THEN
			uiCmdStep:= 0;
		ELSE
			uiCmdStep:= 350;
		END_IF
	END_IF

(* - - - - - - - - - - - - - - - - - - - - - - - - *)
330:(*Set new Min-Level *)
	bSetMinValCmdSt:=FALSE;

	byDTR:=bySetMinValCmdSt;
	IF NOT bActionBusy	THEN
		IF bErr	THEN
			uiCmdStep:= 0;
		ELSE
			uiCmdStep:= 331;
		END_IF
	END_IF

331:(*Set new MinLevel*)
		A_DALICmdSetMinLevel_CmdSt();
	IF NOT bActionBusy	THEN
		IF bErr	THEN
			uiCmdStep:= 0;
		ELSE
			uiCmdStep:= 350;
		END_IF
	END_IF

(* - - - - - - - - - - - - - - - - - - - - - - - - *)
340:(*Set new MaxLevel *)
	bSetMaxValCmdSt:=FALSE;

	byDTR:=bySetMaxValCmdSt;
	IF NOT bActionBusy	THEN
		IF bErr	THEN
			uiCmdStep:= 0;
		ELSE
			uiCmdStep:= 341;
		END_IF
	END_IF

341:(*Set new MaxLevel*)
		A_DALICmdSetMaxLevel_CmdSt();
	IF NOT bActionBusy	THEN
		IF bErr	THEN
			uiCmdStep:= 0;
		ELSE
			uiCmdStep:= 350;
		END_IF
	END_IF

(* - - - - - - - - - - - - - - - - - - - - - - - - *)
(*ZUR SICHERHEIT: ABFRAGE NACH PARAMETRIERUNG*)
350:(*Query Min Level*)
		A_DALICmdQueryMinLevel();
	IF NOT bActionBusy	THEN
		IF bErr	THEN
			uiCmdStep:= 0;
		ELSE
			uiCmdStep:= 351;
		END_IF
	END_IF
	byActlMinCtrlVal:=fbQueryMinLevel.nMinLevel;
	fActlMinCtrlVal := LIMIT(0,LREAL_TO_BYTE(F_fDALICurve(byActlMinCtrlVal)), 254);

351:(*Query Max Level*)
		A_DALICmdQueryMaxLevel();
	IF NOT bActionBusy	THEN
		IF bErr	THEN
			uiCmdStep:= 0;
		ELSE
			uiCmdStep:= 352;
		END_IF
	END_IF
	byActlMaxCtrlVal:=fbQueryMaxLevel.nMaxLevel;
	fActlMaxCtrlVal := F_fDALICurveRev(BYTE_TO_REAL(byActlMaxCtrlVal));

352: (*Lichtabfrage wenn fertig*)
		A_DALICmdQueryActualLevel();
	IF NOT bActionBusy	THEN
		byActlLgtLvl	:= fbQueryActualLevel.nActualLevel;
		uiCmdStep		:= 0;
	END_IF


(* - - - - - - - - - - - - - - - - - - - - - - - - *)
(*Ausschalt-Blinksequenz*)
500: (*Lampe ist bereits aus -> Wartezeit Blinktime*)
	bBusy				:= FALSE;	(*Blinksequenz soll unterbrechbar sein*)
	bBlinkSeqStarted	:= TRUE;
	tonSeqTimer			(IN:= TRUE, PT:=UDINT_TO_TIME(uiBlinkTi*1000));

	IF tonSeqTimer.Q	THEN
		bBusy := TRUE;	(*Verriegelung Kommandoannahme*)
		tonSeqTimer(IN:=FALSE);
		uiCmdStep:= 505;
	END_IF

505: (*Zurück auf ürsprünglich gespeicherten Wert*)
	byArcPowerLevel	:= byRstVal;
		A_DALICmdDirectArcPowerControl();
	IF NOT bActionBusy	THEN
		byActlLgtLvl := byRstVal;
		bBusy:= FALSE;	(*Blinksequenz soll wieder unterbrechbar sein*)
		IF bErr	THEN
			uiCmdStep:= 0;
		ELSE
			uiCmdStep:= 510;
		END_IF
	END_IF

510:(*Wartezeit Off-Delaytime*)
	tonSeqTimer(IN:= TRUE, PT:=UDINT_TO_TIME(uiOffDly*1000));
	IF tonSeqTimer.Q THEN
		bBusy := TRUE;	(*Verriegelung Kommandoannahme*)
		tonSeqTimer(IN:=FALSE);
		uiCmdStep:= 515;
	END_IF

515:(*Off*)
		A_DALICmdOff();
	IF NOT bActionBusy	THEN
		byActlLgtLvl		:= 0;
		bBlinkSeqStarted	:= FALSE;
		bBusy				:= FALSE;
		uiCmdStep			:= 0;
	END_IF

(* - - - - - - - - - - - - - - - - - - - - - - - - *)
(*Init Device-Routine*)

1000: (*Wait fort free DT8*)
	IF NOT arrbBlockDTR[DALI_LINE_NUM] AND g_arrDiagnosisRunOnce[DALI_LINE_NUM] THEN
		uiCmdStep:= 1001;
		arrbBlockDTR[DALI_LINE_NUM]:= TRUE;
		bActionBusy:= FALSE;
	END_IF

1001:(*Set new FadeRate *)
		IF NOT bActionBusy	THEN
			IF bErr	THEN
				uiCmdStep:= 0;
				arrbBlockDTR[DALI_LINE_NUM]:=FALSE;
			ELSE
				uiCmdStep:= 1002;
			END_IF
		END_IF

1002:(*Set new FadeRate*)
	A_DALICmdSetFadeRate();
	IF NOT bActionBusy	THEN
		IF bErr	THEN
			uiCmdStep:= 0;
			arrbBlockDTR[DALI_LINE_NUM]:=FALSE;
		ELSE
			uiCmdStep:= 1003;
		END_IF
	END_IF
	eActlFadeRate:=eFadeRate;

1003:(*Set new FadeTime*)
	eFadeTime_SV:= DALI_Param.eGlobalFadeTime;
	A_DALICmdSetFadeTime();
	IF NOT bActionBusy	THEN
		IF bErr	THEN
			uiCmdStep:= 0;
			arrbBlockDTR[DALI_LINE_NUM]:=FALSE;
		ELSE
			uiCmdStep:= 1010;
		END_IF
	END_IF
	eActlFadeTime:=eFadeTime_SV;
	

1010:(*Set new Min-Level *)
	byDTR:=bySetMinValInput;
	IF NOT bActionBusy	THEN
		IF bErr	THEN
			uiCmdStep:= 0;
			arrbBlockDTR[DALI_LINE_NUM]:=FALSE;
		ELSE
			uiCmdStep:= 1015;
		END_IF
	END_IF

1015:(*Set new Min-Level*)
		A_DALICmdSetMinLevel_Input();
	IF NOT bActionBusy	THEN
		IF bErr	THEN
			uiCmdStep:= 0;
			arrbBlockDTR[DALI_LINE_NUM]:=FALSE;
		ELSE
			uiCmdStep:= 1020;
		END_IF
	END_IF

1020:(*Set new MaxLevel*)
	byDTR:=bySetMaxValInput;
	IF NOT bActionBusy	THEN
		IF bErr	THEN
			uiCmdStep:= 0;
			arrbBlockDTR[DALI_LINE_NUM]:=FALSE;
		ELSE
			uiCmdStep:= 1025;
		END_IF
	END_IF

1025:(*Set new MaxLevel*)
		A_DALICmdSetMaxLevel_Input();
	IF NOT bActionBusy	THEN
		IF bErr	THEN
			uiCmdStep:= 0;
			arrbBlockDTR[DALI_LINE_NUM]:=FALSE;
		ELSE
			uiCmdStep:= 1030;
		END_IF
	END_IF

1030:(*Query physical Min Level*)
		A_DALICmdQueryPhysicalMinLevel();
	IF NOT bActionBusy	THEN
		IF bErr	THEN
			uiCmdStep:= 0;
			arrbBlockDTR[DALI_LINE_NUM]:=FALSE;
		ELSE
			uiCmdStep:= 1035;
		END_IF
	END_IF
	byPhysMinVal:=fbQueryPhysicalMinLevel.nPhysicalMinimum;

1035:(*Query Min Level*)
		A_DALICmdQueryMinLevel();
	IF NOT bActionBusy	THEN
		IF bErr	THEN
			uiCmdStep:= 0;
			arrbBlockDTR[DALI_LINE_NUM]:=FALSE;
		ELSE
			uiCmdStep:= 1040;
		END_IF
	END_IF
	byActlMinCtrlVal:=fbQueryMinLevel.nMinLevel;
	fActlMinCtrlVal := F_fDALICurveRev(BYTE_TO_REAL(byActlMinCtrlVal));

1040:(*Query Max Level*)
		A_DALICmdQueryMaxLevel();
	IF NOT bActionBusy	THEN
		IF bErr	THEN
			uiCmdStep:= 0;
			arrbBlockDTR[DALI_LINE_NUM]:=FALSE;
		ELSE
			uiCmdStep:= 1045;
		END_IF
	END_IF
	byActlMaxCtrlVal:=fbQueryMaxLevel.nMaxLevel;
	fActlMaxCtrlVal := F_fDALICurveRev(BYTE_TO_REAL(byActlMaxCtrlVal));

1045:(*Call Startup-Level*)
	byArcPowerLevel	:= bySttupCtrlVal;
		A_DALICmdDirectArcPowerControl_Sttup();
	IF NOT bActionBusy	THEN
		uiCmdStep:= 1050;
	END_IF

1050: (*Lichtabfrage wenn fertig*)
		A_DALICmdQueryActualLevel();
	IF NOT bActionBusy	THEN
		byActlLgtLvl	:= fbQueryActualLevel.nActualLevel;
		uiCmdStep		:= 0;
		arrbBlockDTR[DALI_LINE_NUM]:=FALSE;
		bInitDone := TRUE;
	END_IF

END_CASE

(*+ + + + + + + + + + + + + + + + + + + + + + + + + + + + + + + + + + + + + + + + + + + + + + + + +*)

IF ((uiPollActLgtLvl > 0) AND (nStepQueryActualLevel = 0) AND (bErr = FALSE)) THEN
	tonCycleActualLevelMasterDev(IN := TRUE, PT := UINT_TO_TIME(uiPollActLgtLvl*1000));
	IF (tonCycleActualLevelMasterDev.Q) THEN
		tonCycleActualLevelMasterDev(IN := FALSE);
		nStepQueryActualLevel := 10;
	END_IF
END_IF

CASE nStepQueryActualLevel OF
0:
	;
10:
	fbQueryActualLevelBackgound(
		bError=> , 
		ipResultMessage=> , 
		bStart:= TRUE, 
		nAddress:= byShrtAdr, 
		eAddressType:= E_DALIAddressType.Short, 
		eCommandPriority:=E_DALICommandPriority.Low , 
		bBusy=> , 
		nActualLevel=> );

	IF (NOT fbQueryActualLevelBackgound.bBusy) THEN
		IF (NOT fbQueryActualLevelBackgound.bError) THEN
			byActlLgtLvl := fbQueryActualLevelBackgound.nActualLevel;
		END_IF
		fbQueryActualLevelBackgound(bStart := FALSE);
		nStepQueryActualLevel := 20;
	END_IF

20:
	fbQueryStatusBackground(
		bError=> , 
		ipResultMessage=> , 
		bStart:= TRUE, 
		nAddress:= byShrtAdr, 
		eAddressType:= E_DALIAddressType.Short, 
		eCommandPriority:= E_DALICommandPriority.Low, 
		bBusy=> , 
		nStatus=> );

	IF (NOT fbQueryStatusBackground.bBusy) THEN
		IF (NOT fbQueryStatusBackground.bError) THEN
			byDALIDevSta := fbQueryStatusBackground.nStatus;
		ELSE
			GVL_DALI_LatestError.arrLineShrtAddr[DALI_LINE_NUM] := byShrtAdr;
		END_IF
		fbQueryStatusBackground(bStart := FALSE);
		nStepQueryActualLevel := 0;
	END_IF
END_CASE

(* + + + + + + + + + + + + + + + + + + + + + + + + + + + + + + + + + + + + + + + + + + + + *)
(*Umrechnung des Lichtwertes lrActlLgtLvl und Speicherung des letzten Wertes vor Aus*)
bLgt			:= BYTE_TO_BOOL		(byActlLgtLvl);
fActlLgtLvl		:= F_fDALICurveRev(BYTE_TO_REAL (byActlLgtLvl));

bMinCtrlValRchd	:= (byActlLgtLvl=byActlMinCtrlVal);
bMaxCtrlValRchd	:= (byActlLgtLvl=byActlMaxCtrlVal);

IF bLgt THEN
	byRstVal:= byActlLgtLvl;
	fRstVal := F_fDALICurveRev(BYTE_TO_REAL(byActlLgtLvl));
END_IF

ACTION A_DALICmdDirectArcPowerControl:
	IF emod = E_DALIAddressType.Group THEN
		byAddr		:= byGrpAdr;
		eAddrType	:= E_DALIAddressType.Group;
	ELSIF emod = E_DALIAddressType.Short THEN
		byAddr		:= byShrtAdr;
		eAddrType	:= E_DALIAddressType.Short;
	END_IF


	bActionBusy	:= TRUE;
	fbDirectArcPowerControl.ipDALICommunication := ipCommunication;

	fbDirectArcPowerControl(
		bError=> , 
		ipResultMessage=> , 
		bStart:=TRUE , 
		nAddress:= byAddr, 
		eAddressType:= eAddrType, 
		eCommandPriority:=Tc3_DALI.E_DALICommandPriority.Middle , 
		bBusy=> , 
		nArcPowerLevel:= byArcPowerLevel);

	IF NOT fbDirectArcPowerControl.bBusy	THEN
		IF	fbDirectArcPowerControl.bError	THEN
			bErr     	:= TRUE;
			nErrorId := fbDirectArcPowerControl.ipResultMessage.nEventId;
		END_IF
		byActlLgtLvl:=byArcPowerLevel;
		bActionBusy		:= FALSE;
		fbDirectArcPowerControl(bStart:= FALSE);
	END_IF
END_ACTION

ACTION A_DALICmdDirectArcPowerControl_Sttup:
	IF emod = E_DALIAddressType.Group THEN
		byAddr		:= byGrpAdr;
		eAddrType	:= E_DALIAddressType.Group;
	ELSIF emod = E_DALIAddressType.Short THEN
		byAddr		:= byShrtAdr;
		eAddrType	:= E_DALIAddressType.Short;
	END_IF

	bActionBusy	:= TRUE;
	

	fbDirectArcPowerControl(
		bError=> , 
		ipResultMessage=> , 
		bStart:=TRUE , 
		nAddress:= byAddr, 
		eAddressType:= eAddrType, 
		eCommandPriority:=Tc3_DALI.E_DALICommandPriority.Middle , 
		bBusy=> , 
		nArcPowerLevel:= byArcPowerLevel);	
	

	IF NOT fbDirectArcPowerControl.bBusy	THEN
		IF	fbDirectArcPowerControl.bError	THEN
			bErr     	:= TRUE;
			nErrorId := fbDirectArcPowerControl.ipResultMessage.nEventId;
		END_IF
		bActionBusy		:= FALSE;
		fbDirectArcPowerControl(bStart:= FALSE);
	END_IF
END_ACTION

ACTION A_DALICmdDown:
	IF emod = E_DALIAddressType.Group THEN
		byAddr		:= byGrpAdr;
		eAddrType	:= E_DALIAddressType.Group;
	ELSIF emod = E_DALIAddressType.Short THEN
		byAddr		:= byShrtAdr;
		eAddrType	:= E_DALIAddressType.Short;
	END_IF

	bActionBusy	:= TRUE;
	
	fbDwn(
		bError=> , 
		ipResultMessage=> , 
		bStart:= TRUE, 
		nAddress:= byAddr, 
		eAddressType:= eAddrType, 
		eCommandPriority:= Tc3_DALI.E_DALICommandPriority.High, 
		bBusy=> );
	
	
	IF NOT fbDwn.bBusy	THEN
		IF	fbDwn.bError	THEN
			bErr     	:= TRUE;
			nErrorId := fbDwn.ipResultMessage.nEventId;
		END_IF
		bActionBusy		:= FALSE;
		fbDwn(bStart:= FALSE);
	END_IF
END_ACTION

ACTION A_DALICmdOff:
	IF emod = E_DALIAddressType.Group THEN
		byAddr		:= byGrpAdr;
		eAddrType	:= E_DALIAddressType.Group;
	ELSIF emod = E_DALIAddressType.Short THEN
		byAddr		:= byShrtAdr;
		eAddrType	:= E_DALIAddressType.Short;
	END_IF


	bActionBusy	:= TRUE;

	fbOff(
		bError=> , 
		ipResultMessage=> , 
		bStart:= TRUE, 
		nAddress:= byAddr, 
		eAddressType:= eAddrType, 
		eCommandPriority:=Tc3_DALI.E_DALICommandPriority.Middle , 
		bBusy=> );
	
	IF NOT fbOff.bBusy	THEN
		IF	fbOff.bError	THEN
			bErr     	:= TRUE;
			nErrorId := fbOff.ipResultMessage.nEventId;

		END_IF
		bActionBusy		:= FALSE;
		fbOff(bStart:= FALSE);
	END_IF
END_ACTION

ACTION A_DALICmdQueryActualLevel:
	bActionBusy	:= TRUE;

	
fbQueryActualLevel(
	bError=> , 
	ipResultMessage=> , 
	bStart:= TRUE, 
	nAddress:= byShrtAdr, 
	eAddressType:= E_DALIAddressType.Short, 
	eCommandPriority:= E_DALICommandPriority.Middle, 
	bBusy=> , 
	nActualLevel=> );

	IF NOT fbQueryActualLevel.bBusy	THEN
		IF	fbQueryActualLevel.bError	THEN
			bErr     	:= TRUE;
			nErrorId := fbQueryActualLevel.ipResultMessage.nEventId;
		END_IF
		bActionBusy		:= FALSE;
		fbQueryActualLevel(bStart:= FALSE );
	END_IF
END_ACTION

ACTION A_DALICmdQueryMaxLevel:
	bActionBusy	:= TRUE;

fbQueryMaxLevel(
	bError=> , 
	ipResultMessage=> , 
	bStart:= TRUE, 
	nAddress:= byShrtAdr, 
	eAddressType:= E_DALIAddressType.Short, 
	eCommandPriority:= E_DALICommandPriority.Middle, 
	bBusy=> , 
	nMaxLevel=> );	
	


	IF NOT fbQueryMaxLevel.bBusy	THEN
		IF	fbQueryMaxLevel.bError	THEN
			bErr     	:= TRUE;
		END_IF
		bActionBusy		:= FALSE;
		fbQueryMaxLevel(bStart:= FALSE);
	END_IF
END_ACTION

ACTION A_DALICmdQueryMinLevel:
	bActionBusy	:= TRUE;

fbQueryMinLevel(
	bError=> , 
	ipResultMessage=> , 
	bStart:= TRUE, 
	nAddress:= byShrtAdr, 
	eAddressType:= E_DALIAddressType.Short, 
	eCommandPriority:= E_DALICommandPriority.Middle, 
	bBusy=> , 
	nMinLevel=> );	

	IF NOT fbQueryMinLevel.bBusy	THEN
		IF	fbQueryMinLevel.bError	THEN
			bErr     	:= TRUE;

		END_IF
		bActionBusy		:= FALSE;
		fbQueryMinLevel(bStart:= FALSE);
	END_IF
END_ACTION

ACTION A_DALICmdQueryPhysicalMinLevel:
	bActionBusy	:= TRUE;

	fbQueryPhysicalMinLevel(
		bError=> , 
		ipResultMessage=> , 
		bStart:= TRUE , 
		nAddress:= byShrtAdr, 
		eAddressType:= E_DALIAddressType.Short, 
		eCommandPriority:= E_DALICommandPriority.Middle, 
		bBusy=> , 
		nPhysicalMinimum=> );


	IF NOT fbQueryPhysicalMinLevel.bBusy	THEN
		IF	fbQueryPhysicalMinLevel.bError	THEN
			bErr     	:= TRUE;

		END_IF
		bActionBusy		:= FALSE;
		fbQueryPhysicalMinLevel(bStart:= FALSE);
	END_IF
END_ACTION

ACTION A_DALICmdRecallMaxLevel:
	IF emod = E_DALIAddressType.Group THEN
		byAddr		:= byGrpAdr;
		eAddrType	:= E_DALIAddressType.Group;
	ELSIF emod = E_DALIAddressType.Short THEN
		byAddr		:= byShrtAdr;
		eAddrType	:= E_DALIAddressType.Short;
	END_IF

	bActionBusy	:= TRUE;

	fbRecallMaxLevel(
		bError=> , 
		ipResultMessage=> , 
		bStart:= TRUE, 
		nAddress:= byAddr, 
		eAddressType:= eAddrType, 
		eCommandPriority:= E_DALICommandPriority.Middle, 
		bBusy=> );


	IF NOT fbRecallMaxLevel.bBusy	THEN
		IF	fbRecallMaxLevel.bError	THEN
			bErr     	:= TRUE;
		END_IF
		bActionBusy		:= FALSE;
		fbRecallMaxLevel(bStart:= FALSE);
	END_IF
END_ACTION

ACTION A_DALICmdRecallMinLevel:
	IF emod = E_DALIAddressType.Group THEN
		byAddr		:= byGrpAdr;
		eAddrType	:= E_DALIAddressType.Group;
	ELSIF emod = E_DALIAddressType.Short THEN
		byAddr		:= byShrtAdr;
		eAddrType	:= E_DALIAddressType.Short;
	END_IF


	bActionBusy	:= TRUE;

	fbRecallMinLevel(
		bError=> , 
		ipResultMessage=> , 
		bStart:= TRUE, 
		nAddress:= byAddr, 
		eAddressType:= eAddrType, 
		eCommandPriority:= E_DALICommandPriority.Middle, 
		bBusy=> );

	IF NOT fbRecallMinLevel.bBusy	THEN
		IF	fbRecallMinLevel.bError	THEN
			bErr     	:= TRUE;

		END_IF
		bActionBusy		:= FALSE;
		fbRecallMinLevel(bStart:= FALSE );
	END_IF
END_ACTION

ACTION A_DALICmdSetFadeRate:
	IF emod = E_DALIAddressType.Group THEN
		byAddr		:= byGrpAdr;
		eAddrType	:= E_DALIAddressType.Group;
	ELSIF emod = E_DALIAddressType.Short THEN
		byAddr		:= byShrtAdr;
		eAddrType	:= E_DALIAddressType.Short;
	END_IF

	bActionBusy	:= TRUE;

	fbSetFadeRate(
		bError=> , 
		ipResultMessage=> , 
		bStart:= TRUE, 
		nAddress:= byAddr , 
		eAddressType:= eAddrType , 
		eCommandPriority:=Tc3_DALI.E_DALICommandPriority.Middle , 
		bBusy=> , 
		eFadeRate:=eFadeRate );
	
	IF (NOT fbSetFadeRate.bBusy) THEN
		IF fbSetFadeRate.bError THEN
			bErr := TRUE;
			nErrorId := fbSetFadeRate.ipResultMessage.nEventId;
		END_IF
		bActionBusy		:= FALSE;
		fbSetFadeRate(bStart:= FALSE);
	END_IF
END_ACTION

ACTION A_DALICmdSetFadeTime:
	IF emod = E_DALIAddressType.Group THEN
		byAddr		:= byGrpAdr;
		eAddrType	:= E_DALIAddressType.Group;
	ELSIF emod = E_DALIAddressType.Short THEN
		byAddr		:= byShrtAdr;
		eAddrType	:= E_DALIAddressType.Short;
	END_IF


	bActionBusy	:= TRUE;

	fbSetFadeTime(
		bError=> , 
		ipResultMessage=> , 
		bStart:= TRUE, 
		nAddress:= byAddr , 
		eAddressType:= eAddrType , 
		eCommandPriority:=Tc3_DALI.E_DALICommandPriority.Middle , 
		bBusy=> , 
		eFadeTime:=eFadeTime_SV );
	
	IF (NOT fbSetFadeTime.bBusy) THEN
		IF fbSetFadeTime.bError THEN
			bErr := TRUE;
			nErrorId := fbSetFadeTime.ipResultMessage.nEventId;
		END_IF
		bActionBusy		:= FALSE;
		fbSetFadeTime(bStart:= FALSE);
	END_IF
END_ACTION

ACTION A_DALICmdSetMaxLevel_CmdSt:


	IF emod = E_DALIAddressType.Group THEN
		byAddr		:= byGrpAdr;
		eAddrType	:= E_DALIAddressType.Group;
	ELSIF emod = E_DALIAddressType.Short THEN
		byAddr		:= byShrtAdr;
		eAddrType	:= E_DALIAddressType.Short;
	END_IF


	bActionBusy	:= TRUE;

	fbSetMaxLevel(
		bError=> , 
		ipResultMessage=> , 
		bStart:= TRUE, 
		nAddress:= byAddr , 
		eAddressType:= eAddrType , 
		eCommandPriority:=Tc3_DALI.E_DALICommandPriority.Middle , 
		bBusy=> , 
		nMaxLevel:= byDTR);
	

	IF (NOT fbSetMaxLevel.bBusy) THEN
		IF fbSetMaxLevel.bError THEN
			bErr := TRUE;
			nErrorId := fbSetMaxLevel.ipResultMessage.nEventId;
		END_IF
		bActionBusy		:= FALSE;
		fbSetMaxLevel(bStart:= FALSE);
	END_IF
END_ACTION

ACTION A_DALICmdSetMaxLevel_Input:


	IF emod = E_DALIAddressType.Group THEN
		byAddr		:= byGrpAdr;
		eAddrType	:= E_DALIAddressType.Group;
	ELSIF emod = E_DALIAddressType.Short THEN
		byAddr		:= byShrtAdr;
		eAddrType	:= E_DALIAddressType.Short;
	END_IF


	bActionBusy	:= TRUE;

	fbSetMaxLevel(
		bError=> , 
		ipResultMessage=> , 
		bStart:= TRUE, 
		nAddress:= byAddr , 
		eAddressType:= eAddrType , 
		eCommandPriority:=Tc3_DALI.E_DALICommandPriority.Middle , 
		bBusy=> , 
		nMaxLevel:= byDTR);
	

	IF (NOT fbSetMaxLevel.bBusy) THEN
		IF fbSetMaxLevel.bError THEN
			bErr := TRUE;
			nErrorId := fbSetMaxLevel.ipResultMessage.nEventId;
		END_IF
		bActionBusy		:= FALSE;
		fbSetMaxLevel(bStart:= FALSE);
	END_IF
END_ACTION

ACTION A_DALICmdSetMinLevel_CmdSt:

	IF emod = E_DALIAddressType.Group THEN
		byAddr		:= byGrpAdr;
		eAddrType	:= E_DALIAddressType.Group;
	ELSIF emod = E_DALIAddressType.Short THEN
		byAddr		:= byShrtAdr;
		eAddrType	:= E_DALIAddressType.Short;
	END_IF


	bActionBusy	:= TRUE;

	fbSetMinLevel(
		bError=> , 
		ipResultMessage=> , 
		bStart:= TRUE, 
		nAddress:= byAddr , 
		eAddressType:= eAddrType , 
		eCommandPriority:=Tc3_DALI.E_DALICommandPriority.Middle , 
		bBusy=> , 
		nMinLevel:= byDTR);
	

	IF (NOT fbSetMinLevel.bBusy) THEN
		IF fbSetMinLevel.bError THEN
			bErr := TRUE;
			nErrorId := fbSetMinLevel.ipResultMessage.nEventId;
		END_IF
		bActionBusy		:= FALSE;
		fbSetMinLevel(bStart:= FALSE);
	END_IF
END_ACTION

